ACTION _brand_colors:
IF csp_main_brand.count = '6Count' 
THEN
	brand1_active := TRUE;
ELSE
	brand1_active := FALSE;
END_IF
IF csp_main_brand.count = '8Count' 
THEN
	brand2_active := TRUE;
ELSE
	brand2_active := FALSE;
END_IF
IF csp_main_brand.count = '10Count' 
THEN
	brand3_active := TRUE;
ELSE
	brand3_active := FALSE;
END_IF
IF csp_main_brand.count = '12Count' 
THEN
	brand4_active := TRUE;
ELSE
	brand4_active := FALSE;
END_IF
IF csp_main_brand.count = '16Count2x3' 
THEN
	brand5_active := TRUE;
ELSE
	brand5_active := FALSE;
END_IF
IF csp_main_brand.count = '18Count' 
THEN
	brand6_active := TRUE;
ELSE
	brand6_active := FALSE;
END_IF
IF csp_main_brand.count = '14Count' 
THEN
	brand7_active := TRUE;
ELSE
	brand7_active := FALSE;
END_IF
IF csp_main_brand.count = '16Count2x4' 
THEN
	brand8_active := TRUE;
ELSE
	brand8_active := FALSE;
END_IF
IF csp_main_brand.count = '20Count' 
THEN
	brand9_active := TRUE;
ELSE
	brand9_active := FALSE;
END_IF
IF csp_main_brand.count = '22Count' 
THEN
	brand10_active := TRUE;
ELSE
	brand10_active := FALSE;
END_IF
IF csp_main_brand.count = '24Count' 
THEN
	brand11_active := TRUE;
ELSE
	brand11_active := FALSE;
END_IF
IF csp_main_brand.count = '28Count' 
THEN
	brand12_active := TRUE;
ELSE
	brand12_active := FALSE;
END_IF
IF csp_main_brand.count = '30Count' 
THEN
	brand13_active := TRUE;
ELSE
	brand13_active := FALSE;
END_IF
IF csp_main_brand.count = '32Count' 
THEN
	brand14_active := TRUE;
ELSE
	brand14_active := FALSE;
END_IF
IF csp_main_brand.count = '34Count' 
THEN
	brand15_active := TRUE;
ELSE
	brand15_active := FALSE;
END_IF
IF csp_main_brand.count = '36Count' 
THEN
	brand16_active := TRUE;
ELSE
	brand16_active := FALSE;
END_IF
IF csp_main_brand.count = '44Count' 
THEN
	brand17_active := TRUE;
ELSE
	brand17_active := FALSE;
END_IF
IF csp_main_brand.count = '46Count' 
THEN
	brand18_active := TRUE;
ELSE
	brand18_active := FALSE;
END_IF
IF csp_main_brand.count = '48Count' 
THEN
	brand19_active := TRUE;
ELSE
	brand19_active := FALSE;
END_IF
IF brand1_active 
THEN
	hmi_change_part_eoat_color := RED;
	hmi_change_part_pusher_color := GREEN;
	hmi_change_part_plate_color	:= GREEN;
	hmi_change_part_paddle_color := RED; (* NO COLOR BUT NEEDS VALUE *)
END_IF
IF brand2_active 
THEN
	hmi_change_part_eoat_color := GREEN;
	hmi_change_part_pusher_color := GREEN;
	hmi_change_part_plate_color	:= GREEN;
	hmi_change_part_paddle_color := RED; (* NO COLOR BUT NEEDS VALUE *)
END_IF
IF brand3_active 
THEN
	hmi_change_part_eoat_color := BLUE;
	hmi_change_part_pusher_color := YELLOW;
	hmi_change_part_plate_color	:= YELLOW;
	hmi_change_part_paddle_color := RED; (* NO COLOR BUT NEEDS VALUE *)
END_IF
IF brand4_active 
THEN
	hmi_change_part_eoat_color := BLUE;
	hmi_change_part_pusher_color := YELLOW;
	hmi_change_part_plate_color	:= YELLOW;
	hmi_change_part_paddle_color := RED; (* NO COLOR BUT NEEDS VALUE *)
END_IF
IF brand5_active 
THEN
	hmi_change_part_eoat_color := BLUE;
	hmi_change_part_pusher_color := YELLOW;
	hmi_change_part_plate_color	:= YELLOW;
	hmi_change_part_paddle_color := RED; (* NO COLOR BUT NEEDS VALUE *)
END_IF
IF brand6_active 
THEN
	hmi_change_part_eoat_color := BLUE;
	hmi_change_part_pusher_color := YELLOW;
	hmi_change_part_plate_color	:= YELLOW;
	hmi_change_part_paddle_color := RED; (* NO COLOR BUT NEEDS VALUE *)
END_IF
IF brand7_active 
THEN
	hmi_change_part_eoat_color := YELLOW;
	hmi_change_part_pusher_color := YELLOW;
	hmi_change_part_plate_color	:= YELLOW;
	hmi_change_part_paddle_color := RED; (* NO COLOR BUT NEEDS VALUE *)
END_IF
IF brand8_active 
THEN
	hmi_change_part_eoat_color := YELLOW;
	hmi_change_part_pusher_color := YELLOW;
	hmi_change_part_plate_color	:= YELLOW;
	hmi_change_part_paddle_color := RED; (* NO COLOR BUT NEEDS VALUE *)
END_IF
IF brand9_active 
THEN
	hmi_change_part_eoat_color := YELLOW;
	hmi_change_part_pusher_color := YELLOW;
	hmi_change_part_plate_color	:= YELLOW;
	hmi_change_part_paddle_color := RED; (* NO COLOR BUT NEEDS VALUE *)
END_IF
IF brand10_active 
THEN
	hmi_change_part_eoat_color := YELLOW;
	hmi_change_part_pusher_color := YELLOW;
	hmi_change_part_plate_color	:= YELLOW;
	hmi_change_part_paddle_color := RED; (* NO COLOR BUT NEEDS VALUE *)
END_IF
IF brand11_active 
THEN
	hmi_change_part_eoat_color := YELLOW;
	hmi_change_part_pusher_color := YELLOW;
	hmi_change_part_plate_color	:= YELLOW;
	hmi_change_part_paddle_color := RED; (* NO COLOR BUT NEEDS VALUE *)
END_IF
IF brand12_active 
THEN
	hmi_change_part_eoat_color := WHITE;
	hmi_change_part_pusher_color := WHITE;
	hmi_change_part_plate_color	:= BLACK;
	hmi_change_part_paddle_color := RED; (* NO COLOR BUT NEEDS VALUE *)
END_IF
IF brand13_active 
THEN
	hmi_change_part_eoat_color := WHITE;
	hmi_change_part_pusher_color := WHITE;
	hmi_change_part_plate_color	:= BLACK;
	hmi_change_part_paddle_color := RED; (* NO COLOR BUT NEEDS VALUE *)
END_IF
IF brand14_active 
THEN
	hmi_change_part_eoat_color := WHITE;
	hmi_change_part_pusher_color := WHITE;
	hmi_change_part_plate_color	:= BLACK;
	hmi_change_part_paddle_color := RED; (* NO COLOR BUT NEEDS VALUE *)
END_IF
IF brand15_active 
THEN
	hmi_change_part_eoat_color := BLACK;
	hmi_change_part_pusher_color := BLACK;
	hmi_change_part_plate_color	:= BLACK;
	hmi_change_part_paddle_color := RED; (* NO COLOR BUT NEEDS VALUE *)
END_IF
IF brand16_active 
THEN
	hmi_change_part_eoat_color := BLACK;
	hmi_change_part_pusher_color := BLACK;
	hmi_change_part_plate_color	:= BLACK;
	hmi_change_part_paddle_color := RED; (* NO COLOR BUT NEEDS VALUE *)
END_IF
IF brand17_active 
THEN
	hmi_change_part_eoat_color := ORANGE;
	hmi_change_part_pusher_color := BLACK;
	hmi_change_part_plate_color	:= BLACK;
	hmi_change_part_paddle_color := RED; (* NO COLOR BUT NEEDS VALUE *)
END_IF
IF brand18_active 
THEN
	hmi_change_part_eoat_color := ORANGE;
	hmi_change_part_pusher_color := BLACK;
	hmi_change_part_plate_color	:= BLACK;
	hmi_change_part_paddle_color := RED; (* NO COLOR BUT NEEDS VALUE *)
END_IF
IF brand19_active 
THEN
	hmi_change_part_eoat_color := RED;		//07/08/21 PRS (was ORANGE)
	hmi_change_part_pusher_color := BLACK;
	hmi_change_part_plate_color	:= BLACK;
	hmi_change_part_paddle_color := RED; (* NO COLOR BUT NEEDS VALUE *)
END_IF
END_ACTION

ACTION _handle_messages:
IF	navigate_to_accU_popup
THEN
	process_message_set(
		errorID_1			:= 0,//fbConfigKinGroup.nErrorId,
		errorID_2			:= 0,
		errorID_3			:= 0,
		CONVERSION_this 	:= navigate_custom_screen_aem);
ELSE
	process_message_reset(navigate_custom_screen_aem);
END_IF

IF	trigger_change_parts_incorrect_popup
THEN
	process_message_set(
		errorID_1			:= 0,
		errorID_2			:= 0,
		errorID_3			:= 0,
		CONVERSION_this 	:= change_parts_incorrect_aem);
ELSE
	process_message_reset(change_parts_incorrect_aem);
END_IF
END_ACTION

ACTION _handle_process_test:
;
END_ACTION

ACTION _hmi_management:
CASE hmi_current_accU_step OF
	0:
		hmi_accU_step1_on:= FALSE;
		hmi_accU_step2_on:= FALSE;
		hmi_accU_step3_on:= FALSE;
		hmi_accU_step4_on:= FALSE;
		hmi_accU_step5_on:= FALSE;
		hmi_accU_step6_on:= FALSE;
		hmi_accU_step7_on:= FALSE;
	1:
		hmi_accU_step1_on:= TRUE;
		hmi_accU_step2_on:= FALSE;
		hmi_accU_step3_on:= FALSE;
		hmi_accU_step4_on:= FALSE;
		hmi_accU_step5_on:= FALSE;
		hmi_accU_step6_on:= FALSE;
		hmi_accU_step7_on:= FALSE;
	2:
		hmi_accU_step1_on:= FALSE;
		hmi_accU_step2_on:= TRUE;
		hmi_accU_step3_on:= FALSE;
		hmi_accU_step4_on:= FALSE;
		hmi_accU_step5_on:= FALSE;
		hmi_accU_step6_on:= FALSE;
		hmi_accU_step7_on:= FALSE;
	3:
		hmi_accU_step1_on:= FALSE;
		hmi_accU_step2_on:= FALSE;
		hmi_accU_step3_on:= TRUE;
		hmi_accU_step4_on:= FALSE;
		hmi_accU_step5_on:= FALSE;
		hmi_accU_step6_on:= FALSE;
		hmi_accU_step7_on:= FALSE;
	4:
		hmi_accU_step1_on:= FALSE;
		hmi_accU_step2_on:= FALSE;
		hmi_accU_step3_on:= FALSE;
		hmi_accU_step4_on:= TRUE;
		hmi_accU_step5_on:= FALSE;
		hmi_accU_step6_on:= FALSE;
		hmi_accU_step7_on:= FALSE;
	5:
		hmi_accU_step1_on:= FALSE;
		hmi_accU_step2_on:= FALSE;
		hmi_accU_step3_on:= FALSE;
		hmi_accU_step4_on:= FALSE;
		hmi_accU_step5_on:= TRUE;
		hmi_accU_step6_on:= FALSE;
		hmi_accU_step7_on:= FALSE;
	6:
		hmi_accU_step1_on:= FALSE;
		hmi_accU_step2_on:= FALSE;
		hmi_accU_step3_on:= FALSE;
		hmi_accU_step4_on:= FALSE;
		hmi_accU_step5_on:= FALSE;
		hmi_accU_step6_on:= TRUE;
		hmi_accU_step7_on:= FALSE;
	7:
		hmi_accU_step1_on:= FALSE;
		hmi_accU_step2_on:= FALSE;
		hmi_accU_step3_on:= FALSE;
		hmi_accU_step4_on:= FALSE;
		hmi_accU_step5_on:= FALSE;
		hmi_accU_step6_on:= FALSE;
		hmi_accU_step7_on:= TRUE;
END_CASE

CASE hmi_change_part_eoat_color OF
	RED:
		hmi_change_part_eoat_red_on:= TRUE;
		hmi_change_part_eoat_green_on:= FALSE;
		hmi_change_part_eoat_blue_on:= FALSE;
		hmi_change_part_eoat_yellow_on:= FALSE;
		hmi_change_part_eoat_white_on:= FALSE;
		hmi_change_part_eoat_black_on:= FALSE;
		hmi_change_part_eoat_orange_on:= FALSE;
	GREEN:
		hmi_change_part_eoat_red_on:= FALSE;
		hmi_change_part_eoat_green_on:= TRUE;
		hmi_change_part_eoat_blue_on:= FALSE;
		hmi_change_part_eoat_yellow_on:= FALSE;
		hmi_change_part_eoat_white_on:= FALSE;
		hmi_change_part_eoat_black_on:= FALSE;
		hmi_change_part_eoat_orange_on:= FALSE;
	BLUE:
		hmi_change_part_eoat_red_on:= FALSE;
		hmi_change_part_eoat_green_on:= FALSE;
		hmi_change_part_eoat_blue_on:= TRUE;
		hmi_change_part_eoat_yellow_on:= FALSE;
		hmi_change_part_eoat_white_on:= FALSE;
		hmi_change_part_eoat_black_on:= FALSE;
		hmi_change_part_eoat_orange_on:= FALSE;
	YELLOW:
		hmi_change_part_eoat_red_on:= FALSE;
		hmi_change_part_eoat_green_on:= FALSE;
		hmi_change_part_eoat_blue_on:= FALSE;
		hmi_change_part_eoat_yellow_on:= TRUE;
		hmi_change_part_eoat_white_on:= FALSE;
		hmi_change_part_eoat_black_on:= FALSE;
		hmi_change_part_eoat_orange_on:= FALSE;
	WHITE:
		hmi_change_part_eoat_red_on:= FALSE;
		hmi_change_part_eoat_green_on:= FALSE;
		hmi_change_part_eoat_blue_on:= FALSE;
		hmi_change_part_eoat_yellow_on:= FALSE;
		hmi_change_part_eoat_white_on:= TRUE;
		hmi_change_part_eoat_black_on:= FALSE;
		hmi_change_part_eoat_orange_on:= FALSE;
	BLACK:
		hmi_change_part_eoat_red_on:= FALSE;
		hmi_change_part_eoat_green_on:= FALSE;
		hmi_change_part_eoat_blue_on:= FALSE;
		hmi_change_part_eoat_yellow_on:= FALSE;
		hmi_change_part_eoat_white_on:= FALSE;
		hmi_change_part_eoat_black_on:= TRUE;
		hmi_change_part_eoat_orange_on:= FALSE;
	ORANGE:
		hmi_change_part_eoat_red_on:= FALSE;
		hmi_change_part_eoat_green_on:= FALSE;
		hmi_change_part_eoat_blue_on:= FALSE;
		hmi_change_part_eoat_yellow_on:= FALSE;
		hmi_change_part_eoat_white_on:= FALSE;
		hmi_change_part_eoat_black_on:= FALSE;
		hmi_change_part_eoat_orange_on:= TRUE;
END_CASE

CASE hmi_change_part_pusher_color OF
	GREEN:
		hmi_change_part_pusher_green_on:= TRUE;
		hmi_change_part_pusher_yellow_on:= FALSE;
		hmi_change_part_pusher_white_on:= FALSE;
		hmi_change_part_pusher_black_on:= FALSE;
	YELLOW:
		hmi_change_part_pusher_green_on:= FALSE;
		hmi_change_part_pusher_yellow_on:= TRUE;
		hmi_change_part_pusher_white_on:= FALSE;
		hmi_change_part_pusher_black_on:= FALSE;
	WHITE:
		hmi_change_part_pusher_green_on:= FALSE;
		hmi_change_part_pusher_yellow_on:= FALSE;
		hmi_change_part_pusher_white_on:= TRUE;
		hmi_change_part_pusher_black_on:= FALSE;
	BLACK:
		hmi_change_part_pusher_green_on:= FALSE;
		hmi_change_part_pusher_yellow_on:= FALSE;
		hmi_change_part_pusher_white_on:= FALSE;
		hmi_change_part_pusher_black_on:= TRUE;
END_CASE

CASE hmi_change_part_plate_color OF
	GREEN:
		hmi_change_part_plate_green_on:= TRUE;
		hmi_change_part_plate_yellow_on:= FALSE;
		hmi_change_part_plate_black_on:= FALSE;
	YELLOW:
		hmi_change_part_plate_green_on:= FALSE;
		hmi_change_part_plate_yellow_on:= TRUE;
		hmi_change_part_plate_black_on:= FALSE;
	BLACK:
		hmi_change_part_plate_green_on:= FALSE;
		hmi_change_part_plate_yellow_on:= FALSE;
		hmi_change_part_plate_black_on:= TRUE;
END_CASE

CASE hmi_change_part_paddle_color OF
	NO_COLOR:
		//FUTURE PLACEHOLDER
END_CASE

	hmi_graphic_object_set_status(
		status  			:= SEL(machine_size_complete, HMI_OBJECT_STATUS_INVISIBLE, HMI_OBJECT_STATUS_ON),
		CONVERSION_this    	:= hmi_brand_status_color_hgos);
	
	hmi_graphic_object_set_status(
		status  			:= SEL(machine_size_complete, HMI_OBJECT_STATUS_ON, HMI_OBJECT_STATUS_INVISIBLE),
		CONVERSION_this    	:= hmi_brand_status_bad_color_hgos);
	
	hmi_graphic_object_set_status(
        status  			:= SEL(hmi_accU_step1_on, HMI_OBJECT_STATUS_INVISIBLE, HMI_OBJECT_STATUS_ON),
        CONVERSION_this     := hmi_accU_step1_on_hgos);
		
	hmi_graphic_object_set_status(
        status  			:= SEL(hmi_accU_step1_on, HMI_OBJECT_STATUS_ON, HMI_OBJECT_STATUS_INVISIBLE),
        CONVERSION_this     := hmi_accU_step1_off_hgos);
		
	hmi_graphic_object_set_status(
        status  			:= SEL(hmi_accU_step2_on, HMI_OBJECT_STATUS_INVISIBLE, HMI_OBJECT_STATUS_ON),
        CONVERSION_this     := hmi_accU_step2_on_hgos);
		
	hmi_graphic_object_set_status(
        status  			:= SEL(hmi_accU_step2_on, HMI_OBJECT_STATUS_ON, HMI_OBJECT_STATUS_INVISIBLE),
        CONVERSION_this     := hmi_accU_step2_off_hgos);
		
	hmi_graphic_object_set_status(
        status  			:= SEL(hmi_accU_step3_on, HMI_OBJECT_STATUS_INVISIBLE, HMI_OBJECT_STATUS_ON),
        CONVERSION_this     := hmi_accU_step3_on_hgos);
		
	hmi_graphic_object_set_status(
        status  			:= SEL(hmi_accU_step3_on, HMI_OBJECT_STATUS_ON, HMI_OBJECT_STATUS_INVISIBLE),
        CONVERSION_this     := hmi_accU_step3_off_hgos);
		
	hmi_graphic_object_set_status(
        status  			:= SEL(hmi_accU_step4_on, HMI_OBJECT_STATUS_INVISIBLE, HMI_OBJECT_STATUS_ON),
        CONVERSION_this     := hmi_accU_step4_on_hgos);
		
	hmi_graphic_object_set_status(
		status  			:= SEL(hmi_accU_step4_on, HMI_OBJECT_STATUS_ON, HMI_OBJECT_STATUS_INVISIBLE),
        CONVERSION_this     := hmi_accU_step4_off_hgos);
		
	hmi_graphic_object_set_status(
        status  			:= SEL(hmi_accU_step5_on, HMI_OBJECT_STATUS_INVISIBLE, HMI_OBJECT_STATUS_ON),
        CONVERSION_this     := hmi_accU_step5_on_hgos);
		
	hmi_graphic_object_set_status(
        status  			:= SEL(hmi_accU_step5_on, HMI_OBJECT_STATUS_ON, HMI_OBJECT_STATUS_INVISIBLE),
        CONVERSION_this     := hmi_accU_step5_off_hgos);
		
	hmi_graphic_object_set_status(
        status  			:= SEL(hmi_accU_step6_on, HMI_OBJECT_STATUS_INVISIBLE, HMI_OBJECT_STATUS_ON),
        CONVERSION_this     := hmi_accU_step6_on_hgos);
		
	hmi_graphic_object_set_status(
        status  			:= SEL(hmi_accU_step6_on, HMI_OBJECT_STATUS_ON, HMI_OBJECT_STATUS_INVISIBLE),
        CONVERSION_this     := hmi_accU_step6_off_hgos);
		
	hmi_graphic_object_set_status(
        status  			:= SEL(hmi_accU_step7_on, HMI_OBJECT_STATUS_INVISIBLE, HMI_OBJECT_STATUS_ON),
        CONVERSION_this     := hmi_accU_step7_on_hgos);
	
	hmi_graphic_object_set_status(
        status  			:= SEL(hmi_accU_step7_on, HMI_OBJECT_STATUS_ON, HMI_OBJECT_STATUS_INVISIBLE),
        CONVERSION_this     := hmi_accU_step7_off_hgos);

	//Change Part EOAT
	hmi_graphic_object_set_status(
        status  			:= SEL(hmi_change_part_eoat_red_on, HMI_OBJECT_STATUS_INVISIBLE, HMI_OBJECT_STATUS_ON),
        CONVERSION_this     := hmi_change_part_eoat_red_hgos);
		
	hmi_graphic_object_set_status(
        status  			:= SEL(hmi_change_part_eoat_green_on, HMI_OBJECT_STATUS_INVISIBLE, HMI_OBJECT_STATUS_ON),
        CONVERSION_this     := hmi_change_part_eoat_green_hgos);
		
	hmi_graphic_object_set_status(
        status  			:= SEL(hmi_change_part_eoat_blue_on, HMI_OBJECT_STATUS_INVISIBLE, HMI_OBJECT_STATUS_ON),
        CONVERSION_this     := hmi_change_part_eoat_blue_hgos);
		
	hmi_graphic_object_set_status(
        status  			:= SEL(hmi_change_part_eoat_yellow_on, HMI_OBJECT_STATUS_INVISIBLE, HMI_OBJECT_STATUS_ON),
        CONVERSION_this     := hmi_change_part_eoat_yellow_hgos);
	
	hmi_graphic_object_set_status(
        status  			:= SEL(hmi_change_part_eoat_white_on, HMI_OBJECT_STATUS_INVISIBLE, HMI_OBJECT_STATUS_ON),
        CONVERSION_this     := hmi_change_part_eoat_white_hgos);
		
	hmi_graphic_object_set_status(
        status  			:= SEL(hmi_change_part_eoat_black_on, HMI_OBJECT_STATUS_INVISIBLE, HMI_OBJECT_STATUS_ON),
        CONVERSION_this     := hmi_change_part_eoat_black_hgos);
		
	hmi_graphic_object_set_status(
        status  			:= SEL(hmi_change_part_eoat_orange_on, HMI_OBJECT_STATUS_INVISIBLE, HMI_OBJECT_STATUS_ON),
        CONVERSION_this     := hmi_change_part_eoat_orange_hgos);
		
	hmi_graphic_object_set_status(
        status  			:= SEL(hmi_change_part_eoat_checkbox_on, HMI_OBJECT_STATUS_INVISIBLE, HMI_OBJECT_STATUS_ON),
        CONVERSION_this     := hmi_change_part_eoat_checkbox_hgos);
		
	//Change Part Pusher
	hmi_graphic_object_set_status(
        status  			:= SEL(hmi_change_part_pusher_green_on, HMI_OBJECT_STATUS_INVISIBLE, HMI_OBJECT_STATUS_ON),
        CONVERSION_this     := hmi_change_part_pusher_green_hgos);
		
	hmi_graphic_object_set_status(
        status  			:= SEL(hmi_change_part_pusher_yellow_on, HMI_OBJECT_STATUS_INVISIBLE, HMI_OBJECT_STATUS_ON),
        CONVERSION_this     := hmi_change_part_pusher_yellow_hgos);
		
	hmi_graphic_object_set_status(
        status  			:= SEL(hmi_change_part_pusher_white_on, HMI_OBJECT_STATUS_INVISIBLE, HMI_OBJECT_STATUS_ON),
        CONVERSION_this     := hmi_change_part_pusher_white_hgos);
		
	hmi_graphic_object_set_status(
        status  			:= SEL(hmi_change_part_pusher_black_on, HMI_OBJECT_STATUS_INVISIBLE, HMI_OBJECT_STATUS_ON),
        CONVERSION_this     := hmi_change_part_pusher_black_hgos);
		
	hmi_graphic_object_set_status(
        status  			:= SEL(hmi_change_part_pusher_checkbox_on, HMI_OBJECT_STATUS_INVISIBLE, HMI_OBJECT_STATUS_ON),
        CONVERSION_this     := hmi_change_part_pusher_checkbox_hgos);
		
	//Change Part Plate
	hmi_graphic_object_set_status(
        status  			:= SEL(hmi_change_part_plate_green_on, HMI_OBJECT_STATUS_INVISIBLE, HMI_OBJECT_STATUS_ON),
        CONVERSION_this     := hmi_change_part_plate_green_hgos);
		
	hmi_graphic_object_set_status(
        status  			:= SEL(hmi_change_part_plate_yellow_on, HMI_OBJECT_STATUS_INVISIBLE, HMI_OBJECT_STATUS_ON),
        CONVERSION_this     := hmi_change_part_plate_yellow_hgos);
		
	hmi_graphic_object_set_status(
        status  			:= SEL(hmi_change_part_plate_black_on, HMI_OBJECT_STATUS_INVISIBLE, HMI_OBJECT_STATUS_ON),
        CONVERSION_this     := hmi_change_part_plate_black_hgos);
		
	hmi_graphic_object_set_status(
        status  			:= SEL(hmi_change_part_plate_checkbox_on, HMI_OBJECT_STATUS_INVISIBLE, HMI_OBJECT_STATUS_ON),
        CONVERSION_this     := hmi_change_part_plate_checkbox_hgos);
	
	//Change Part Paddles
	hmi_graphic_object_set_status(
        status  			:= SEL(hmi_change_part_paddle_checkbox_on, HMI_OBJECT_STATUS_INVISIBLE, HMI_OBJECT_STATUS_ON),
        CONVERSION_this     := hmi_change_part_paddle_checkbox_hgos);
END_ACTION

ACTION _in_position:
IF (csp_case_main_statistics.is_empty
	AND csp_transfer_main_statistics.is_empty 
	AND NOT digital_input_is_active(csp_case_feed_magazine_ls_pusher.retracted_di)
	AND NOT digital_input_is_active(csp_case_feed_magazine_ls_pusherTilt.upstream_di)
	AND NOT digital_input_is_active(csp_case_feed_magazine_os_pusher.retracted_di)
	AND NOT digital_input_is_active(csp_case_feed_magazine_os_pusherTilt.upstream_di)
	AND NOT digital_input_is_active(csp_case_feed_magazine_level_zonemin.di)
	AND NOT digital_input_is_active(csp_case_feed_magazine_level_zonelow.di)
	AND NOT digital_input_is_active(csp_case_feed_magazine_level_zone1.di)
	AND NOT digital_input_is_active(csp_case_feed_magazine_level_zone2.di)
	AND NOT digital_input_is_active(csp_case_feed_magazine_level_zone3.di))
	OR manual_empty
THEN
	machine_empty := TRUE;
ELSE
	machine_empty := FALSE;
END_IF

IF (csp_case_tr_squaring_ls_leading.in_accu_safe_pos)
    AND (csp_case_tr_squaring_ls_trailing.in_accu_safe_pos)
    AND (csp_case_tr_squaring_os_leading.in_accu_safe_pos)
    AND (csp_case_tr_squaring_os_trailing.in_accu_safe_pos)
    AND (csp_case_closing_os_horizontal.in_accu_safe_pos)
    AND (csp_case_closing_os_upper.in_accu_safe_pos)
    AND (csp_case_closing_os_lower.in_accu_safe_pos)
    AND (csp_case_closing_ls_horizontal.in_accu_safe_pos)
    AND (csp_case_closing_ls_upper.in_accu_safe_pos)
    AND (csp_case_closing_ls_lower.in_accu_safe_pos)
    AND (csp_case_fc_ls_lower_follower.in_accu_safe_pos)
    AND (csp_case_fc_ls_lower_spreader.in_accu_safe_pos)
    AND (csp_case_fc_ls_upper_follower.in_accu_safe_pos)
    AND (csp_case_fc_ls_upper_leadingMinorCloser.in_accu_safe_pos)
    AND (csp_case_fc_ls_upper_spreader.in_accu_safe_pos)
    AND (csp_case_fc_os_lower_follower.in_accu_safe_pos)
    AND (csp_case_fc_os_lower_spreader.in_accu_safe_pos)
    AND (csp_case_fc_os_upper_follower.in_accu_safe_pos)
    AND (csp_case_fc_os_upper_spreader.in_accu_safe_pos)
    AND (csp_case_feed_shuttle_vertical.in_accu_safe_pos)
    AND (csp_case_loader_guide_downstream.in_accu_safe_pos)
    AND (csp_case_loader_guide_length.in_accu_safe_pos)
    AND (csp_case_loader_guide_upstream.in_accu_safe_pos)
    AND (csp_case_loader_pusher.in_accu_safe_pos)
	AND (csp_case_feed_kinematic_x.in_accu_safe_pos)
	AND (csp_case_feed_kinematic_y.in_accu_safe_pos)
	AND (csp_case_feed_kinematic_tilt.in_accu_safe_pos) 
THEN
    Case_Motors_Safe_accU := TRUE;
ELSE
    Case_Motors_Safe_accU := FALSE;   
END_IF

	
IF csp_case_feed_shuttle_accU_depth.in_position
	AND csp_case_transport_accU_depth.in_position
	AND csp_case_feed_reject_accU_depth.in_position
THEN
	test_in_position := TRUE;
ELSE
	test_in_position := FALSE;
END_IF

//INSERT IF STATEMENT HERE FOR WHICH MOTORS BELONG TO WHICH GROUP

//Group 1 Motors in Position
IF 	csp_case_transport_accU_depth.in_position
	AND csp_case_feed_shuttle_accU_depth.in_position
	AND csp_case_feed_magazine_accU_lsDepth.in_position
	AND csp_case_feed_magazine_accU_osDepth.in_position
	AND csp_case_feed_reject_accU_depth.in_position
	AND csp_transfer_infeed_accU_depth.in_position
	AND csp_transfer_infeed_accU_waterfallAdjust.in_position
	AND csp_transfer_accumulator_accU_depth.in_position
	AND csp_transfer_accumulator_accU_convDepth.in_position
	AND csp_case_tr_accU_depth.in_position
THEN
	Group_1_motors_in_position := TRUE;
ELSE
	Group_1_motors_in_position := FALSE;
END_IF

//Group 2 Motors in Position
IF 	csp_case_loader_guide_accU_width.in_position
	AND csp_case_glue_os_accU_width.in_position
	AND csp_case_glue_os_accU_upperPosition.in_position
	AND csp_case_glue_os_accU_lowerPosition.in_position
	AND csp_case_glue_ls_accU_upperPosition.in_position
	AND csp_case_glue_ls_accU_lowerPosition.in_position
	AND csp_case_tr_accU_os_width.in_position
	AND csp_case_tr_accU_ls_width.in_position
THEN
	Group_2_motors_in_position := TRUE;
ELSE
	Group_2_motors_in_position := FALSE;
END_IF

IF Case_Motors_In_New_Accu_Pos //AND Transfer_Motors_In_New_Accu_Pos
THEN
	Motion_motors_in_position := TRUE;
ELSE
	Motion_motors_in_position := FALSE;
END_IF


IF 	ABS(csp_case_closing_os_horizontal.axis.actual_position - csp_case_closing_os_horizontal.accu_safe_pos) < csp_case_closing_os_horizontal.accu_tolerance
	AND ABS(csp_case_closing_ls_horizontal.axis.actual_position - csp_case_closing_ls_horizontal.accu_safe_pos) < csp_case_closing_ls_horizontal.accu_tolerance
THEN
	closing_horizontal_safe := TRUE;
ELSE
	closing_horizontal_safe := FALSE;
END_IF


(* Acc U Change indicators on Acc U Change Motor page *)
	
	hmi_graphic_object_set_status(
        status  			:= SEL(csp_case_transport_accU_depth.in_position, HMI_OBJECT_STATUS_INVISIBLE, HMI_OBJECT_STATUS_ON),
        CONVERSION_this     := hmi_in_position_transport_depth_on_hgos);
		
	hmi_graphic_object_set_status(
        status  			:= SEL(csp_case_transport_accU_depth.in_position, HMI_OBJECT_STATUS_ON, HMI_OBJECT_STATUS_INVISIBLE),
        CONVERSION_this     := hmi_in_position_transport_depth_off_hgos);
	
	hmi_graphic_object_set_status(
        status  			:= SEL(csp_case_feed_shuttle_accU_depth.in_position, HMI_OBJECT_STATUS_INVISIBLE, HMI_OBJECT_STATUS_ON),
        CONVERSION_this     := hmi_in_position_shuttle_depth_on_hgos);
		
	hmi_graphic_object_set_status(
        status  			:= SEL(csp_case_feed_shuttle_accU_depth.in_position, HMI_OBJECT_STATUS_ON, HMI_OBJECT_STATUS_INVISIBLE),
        CONVERSION_this     := hmi_in_position_shuttle_depth_off_hgos);

 	hmi_graphic_object_set_status(
        status  			:= SEL(csp_case_feed_magazine_accU_lsDepth.in_position, HMI_OBJECT_STATUS_INVISIBLE, HMI_OBJECT_STATUS_ON),
        CONVERSION_this     := hmi_in_position_magazine_ls_depth_on_hgos);
		
	hmi_graphic_object_set_status(
        status  			:= SEL(csp_case_feed_magazine_accU_lsDepth.in_position, HMI_OBJECT_STATUS_ON, HMI_OBJECT_STATUS_INVISIBLE),
        CONVERSION_this     := hmi_in_position_magazine_ls_depth_off_hgos);
		
	hmi_graphic_object_set_status(
        status  			:= SEL(csp_case_feed_magazine_accU_osDepth.in_position, HMI_OBJECT_STATUS_INVISIBLE, HMI_OBJECT_STATUS_ON),
        CONVERSION_this     := hmi_in_position_magazine_os_depth_on_hgos);
		
	hmi_graphic_object_set_status(
        status  			:= SEL(csp_case_feed_magazine_accU_osDepth.in_position, HMI_OBJECT_STATUS_ON, HMI_OBJECT_STATUS_INVISIBLE),
        CONVERSION_this     := hmi_in_position_magazine_os_depth_off_hgos);
	
	hmi_graphic_object_set_status(
        status  			:= SEL(csp_case_feed_reject_accU_depth.in_position, HMI_OBJECT_STATUS_INVISIBLE, HMI_OBJECT_STATUS_ON),
        CONVERSION_this     := hmi_in_position_discharge_os_depth_on_hgos);
		
	hmi_graphic_object_set_status(
        status  			:= SEL(csp_case_feed_reject_accU_depth.in_position, HMI_OBJECT_STATUS_ON, HMI_OBJECT_STATUS_INVISIBLE),
        CONVERSION_this     := hmi_in_position_discharge_os_depth_off_hgos);
	
	hmi_graphic_object_set_status(
        status  			:= SEL(csp_transfer_infeed_accU_depth.in_position, HMI_OBJECT_STATUS_INVISIBLE, HMI_OBJECT_STATUS_ON),
        CONVERSION_this     := hmi_in_position_transfer_infeed_depth_on_hgos);
		
	hmi_graphic_object_set_status(
        status  			:= SEL(csp_transfer_infeed_accU_depth.in_position, HMI_OBJECT_STATUS_ON, HMI_OBJECT_STATUS_INVISIBLE),
        CONVERSION_this     := hmi_in_position_transfer_infeed_depth_off_hgos);	
		
	hmi_graphic_object_set_status(
        status  			:= SEL(csp_transfer_infeed_accU_waterfallAdjust.in_position, HMI_OBJECT_STATUS_INVISIBLE, HMI_OBJECT_STATUS_ON),
        CONVERSION_this     := hmi_in_position_waterfall_on_hgos);
		
	hmi_graphic_object_set_status(
        status  			:= SEL(csp_transfer_infeed_accU_waterfallAdjust.in_position, HMI_OBJECT_STATUS_ON, HMI_OBJECT_STATUS_INVISIBLE),
        CONVERSION_this     := hmi_in_position_waterfall_off_hgos);	
	 
	hmi_graphic_object_set_status(
        status  			:= SEL(csp_transfer_accumulator_accU_depth.in_position, HMI_OBJECT_STATUS_INVISIBLE, HMI_OBJECT_STATUS_ON),
        CONVERSION_this     := hmi_in_position_accumulator_depth_on_hgos);
		
	hmi_graphic_object_set_status(
        status  			:= SEL(csp_transfer_accumulator_accU_depth.in_position, HMI_OBJECT_STATUS_ON, HMI_OBJECT_STATUS_INVISIBLE),
        CONVERSION_this     := hmi_in_position_accumulator_depth_off_hgos);	
		
	hmi_graphic_object_set_status(
        status  			:= SEL(csp_transfer_accumulator_accU_convDepth.in_position, HMI_OBJECT_STATUS_INVISIBLE, HMI_OBJECT_STATUS_ON),
        CONVERSION_this     := hmi_in_position_accumulator_conv_depth_on_hgos);
		
	hmi_graphic_object_set_status(
        status  			:= SEL(csp_transfer_accumulator_accU_convDepth.in_position, HMI_OBJECT_STATUS_ON, HMI_OBJECT_STATUS_INVISIBLE),
        CONVERSION_this     := hmi_in_position_accumulator_conv_depth_off_hgos);		

	hmi_graphic_object_set_status(
        status  			:= SEL(csp_case_tr_accU_depth.in_position, HMI_OBJECT_STATUS_INVISIBLE, HMI_OBJECT_STATUS_ON),
        CONVERSION_this     := hmi_in_position_top_rail_depth_on_hgos);
		
	hmi_graphic_object_set_status(
        status  			:= SEL(csp_case_tr_accU_depth.in_position, HMI_OBJECT_STATUS_ON, HMI_OBJECT_STATUS_INVISIBLE),
        CONVERSION_this     := hmi_in_position_top_rail_depth_off_hgos);		

	

//Group 2 Motors in Position Acc U Change motor indicators
	hmi_graphic_object_set_status(
        status  			:= SEL(csp_case_loader_guide_accU_width.in_position, HMI_OBJECT_STATUS_INVISIBLE, HMI_OBJECT_STATUS_ON),
        CONVERSION_this     := hmi_in_position_loader_guide_width_on_hgos);
		
	hmi_graphic_object_set_status(
        status  			:= SEL(csp_case_loader_guide_accU_width.in_position, HMI_OBJECT_STATUS_ON, HMI_OBJECT_STATUS_INVISIBLE),
        CONVERSION_this     := hmi_in_position_loader_guide_width_off_hgos);	
	
	hmi_graphic_object_set_status(
        status  			:= SEL(csp_case_glue_os_accU_width.in_position, HMI_OBJECT_STATUS_INVISIBLE, HMI_OBJECT_STATUS_ON),
        CONVERSION_this     := hmi_in_position_glue_os_width_on_hgos);
		
	hmi_graphic_object_set_status(
        status  			:= SEL(csp_case_glue_os_accU_width.in_position, HMI_OBJECT_STATUS_ON, HMI_OBJECT_STATUS_INVISIBLE),
        CONVERSION_this     := hmi_in_position_glue_os_width_off_hgos);	
		
	hmi_graphic_object_set_status(
        status  			:= SEL(csp_case_glue_os_accU_upperPosition.in_position, HMI_OBJECT_STATUS_INVISIBLE, HMI_OBJECT_STATUS_ON),
        CONVERSION_this     := hmi_in_position_glue_os_upper_on_hgos);
		
	hmi_graphic_object_set_status(
        status  			:= SEL(csp_case_glue_os_accU_upperPosition.in_position, HMI_OBJECT_STATUS_ON, HMI_OBJECT_STATUS_INVISIBLE),
        CONVERSION_this     := hmi_in_position_glue_os_upper_off_hgos);	
		
	hmi_graphic_object_set_status(
        status  			:= SEL(csp_case_glue_os_accU_lowerPosition.in_position, HMI_OBJECT_STATUS_INVISIBLE, HMI_OBJECT_STATUS_ON),
        CONVERSION_this     := hmi_in_position_glue_os_lower_on_hgos);
		
	hmi_graphic_object_set_status(
        status  			:= SEL(csp_case_glue_os_accU_lowerPosition.in_position, HMI_OBJECT_STATUS_ON, HMI_OBJECT_STATUS_INVISIBLE),
        CONVERSION_this     := hmi_in_position_glue_os_lower_off_hgos);	
	
	hmi_graphic_object_set_status(
        status  			:= SEL(csp_case_glue_ls_accU_upperPosition.in_position, HMI_OBJECT_STATUS_INVISIBLE, HMI_OBJECT_STATUS_ON),
        CONVERSION_this     := hmi_in_position_glue_ls_upper_on_hgos);
		
	hmi_graphic_object_set_status(
        status  			:= SEL(csp_case_glue_ls_accU_upperPosition.in_position, HMI_OBJECT_STATUS_ON, HMI_OBJECT_STATUS_INVISIBLE),
        CONVERSION_this     := hmi_in_position_glue_ls_upper_off_hgos);	
		
	hmi_graphic_object_set_status(
        status  			:= SEL(csp_case_glue_ls_accU_lowerPosition.in_position, HMI_OBJECT_STATUS_INVISIBLE, HMI_OBJECT_STATUS_ON),
        CONVERSION_this     := hmi_in_position_glue_ls_lower_on_hgos);
		
	hmi_graphic_object_set_status(
        status  			:= SEL(csp_case_glue_ls_accU_lowerPosition.in_position, HMI_OBJECT_STATUS_ON, HMI_OBJECT_STATUS_INVISIBLE),
        CONVERSION_this     := hmi_in_position_glue_ls_lower_off_hgos);	
	
	hmi_graphic_object_set_status(
        status  			:= SEL(csp_case_tr_accU_os_width.in_position, HMI_OBJECT_STATUS_INVISIBLE, HMI_OBJECT_STATUS_ON),
        CONVERSION_this     := hmi_in_position_top_rail_os_width_on_hgos);
		
	hmi_graphic_object_set_status(
        status  			:= SEL(csp_case_tr_accU_os_width.in_position, HMI_OBJECT_STATUS_ON, HMI_OBJECT_STATUS_INVISIBLE),
        CONVERSION_this     := hmi_in_position_top_rail_os_width_off_hgos);	


	hmi_graphic_object_set_status(
        status  			:= SEL(csp_case_tr_accU_ls_width.in_position, HMI_OBJECT_STATUS_INVISIBLE, HMI_OBJECT_STATUS_ON),
        CONVERSION_this     := hmi_in_position_top_rail_ls_width_on_hgos);
		
	hmi_graphic_object_set_status(
        status  			:= SEL(csp_case_tr_accU_ls_width.in_position, HMI_OBJECT_STATUS_ON, HMI_OBJECT_STATUS_INVISIBLE),
        CONVERSION_this     := hmi_in_position_top_rail_ls_width_off_hgos);
END_ACTION

ACTION _mode_manager:
IF process_mode_req_is_pending(prc)
THEN
    process_apply_mode_req_first_step(prc);
    CASE process_get_mode(prc) OF
        MODE_TO_ABSENT:
			;
        MODE_TO_INACTIVE:
			;
        MODE_TO_TEST:
			;
        MODE_TO_OPERATIONAL:
			;
    END_CASE
    process_apply_mode_req_second_step(prc);
END_IF
END_ACTION

ACTION _object_manager:
IF objects_initialization()
THEN
	sub_process_init(
		object_name					:= 'csp_main_accuChange.prc', 
		process						:= csp_main.prc, 
		CONVERSION_this				:= prc);
		
	prc_path 						:= process_get_path(prc);
	
	process_message_init(
		object_name					:= CONCAT(prc_path, '_navigate_custom_screen_aem'), 
		behaviour					:= MESSAGE_BEHAVIOUR_STATE,
		reset_timeout				:= 0,
		disableable					:= FALSE,
		individual_reset			:= FALSE,
		machine_reaction			:= MACHINE_REACTION_NO_STOP,
		typology					:= MESSAGE_TYPOLOGY_OBLIGATION,
		process						:= prc,
		CONVERSION_this				:= navigate_custom_screen_aem);
		
	process_message_init(
		object_name					:= CONCAT(prc_path, '_change_parts_incorrect_aem'), 
		behaviour					:= MESSAGE_BEHAVIOUR_STATE,
		reset_timeout				:= 0,
		disableable					:= FALSE,
		individual_reset			:= FALSE,
		machine_reaction			:= MACHINE_REACTION_NO_STOP,
		typology					:= MESSAGE_TYPOLOGY_OBLIGATION,
		process						:= prc,
		CONVERSION_this				:= change_parts_incorrect_aem);		
		
	timer_init(
		object_name					:= CONCAT(prc_path, '_RFID_read_write_tmr'),
		process						:= prc,
		CONVERSION_this				:= RFID_read_write_tmr);
	
	motorization_conditioner_init(
		object_name					:=	CONCAT(prc_path, 'all_in_position_motcond'),
		velocity_limit				:=	0.0,
		velocity_limit_active		:=	FALSE,
		idle_handshake_active		:=	FALSE,
		execute_handshake_active	:=	TRUE,
		hold_handshake_active		:=	FALSE,
		suspend_handshake_active	:=	FALSE,
		complete_handshake_active	:=	FALSE,
		abort_handshake_active		:=	FALSE,
		stop_handshake_active		:=	FALSE,
		origin						:=	MOTORIZATION_CONDITIONER_ORIGIN_INTERNAL,
		manager						:=	csp_main_motorization_manager.motm,
		process						:=	prc,
		CONVERSION_this				:=	all_in_position_motcond);
		
		
	motorization_conditioner_init(
		object_name					:=	CONCAT(prc_path, '_eoat_rfid_checked_motcond'),
		velocity_limit				:=	0.0,
		velocity_limit_active		:=	FALSE,
		idle_handshake_active		:=	FALSE,
		execute_handshake_active	:=	TRUE,
		hold_handshake_active		:=	FALSE,
		suspend_handshake_active	:=	FALSE,
		complete_handshake_active	:=	FALSE,
		abort_handshake_active		:=	FALSE,
		stop_handshake_active		:=	FALSE,
		origin						:=	MOTORIZATION_CONDITIONER_ORIGIN_INTERNAL,
		manager						:=	csp_main_motorization_manager.motm,
		process						:=	prc,
		CONVERSION_this				:=	eoat_rfid_checked_motcond);
		
	motorization_conditioner_init(
		object_name					:=	CONCAT(prc_path, '_loader_pusher_rfid_checked_motcond'),
		velocity_limit				:=	0.0,
		velocity_limit_active		:=	FALSE,
		idle_handshake_active		:=	FALSE,
		execute_handshake_active	:=	TRUE,
		hold_handshake_active		:=	FALSE,
		suspend_handshake_active	:=	FALSE,
		complete_handshake_active	:=	FALSE,
		abort_handshake_active		:=	FALSE,
		stop_handshake_active		:=	FALSE,
		origin						:=	MOTORIZATION_CONDITIONER_ORIGIN_INTERNAL,
		manager						:=	csp_main_motorization_manager.motm,
		process						:=	prc,
		CONVERSION_this				:=	loader_pusher_rfid_checked_motcond);
		
	motorization_conditioner_init(
		object_name					:=	CONCAT(prc_path, '_loader_plate_rfid_checked_motcond'),
		velocity_limit				:=	0.0,
		velocity_limit_active		:=	FALSE,
		idle_handshake_active		:=	FALSE,
		execute_handshake_active	:=	TRUE,
		hold_handshake_active		:=	FALSE,
		suspend_handshake_active	:=	FALSE,
		complete_handshake_active	:=	FALSE,
		abort_handshake_active		:=	FALSE,
		stop_handshake_active		:=	FALSE,
		origin						:=	MOTORIZATION_CONDITIONER_ORIGIN_INTERNAL,
		manager						:=	csp_main_motorization_manager.motm,
		process						:=	prc,
		CONVERSION_this				:=	loader_plate_rfid_checked_motcond);
		
		
	boolean_init(
		object_name:= CONCAT(prc_path, '_motors_in_safe_pos_boolean'), 
		process:= prc, 
		CONVERSION_this:= motors_in_safe_pos_boolean);
		
	digital_check_and_message_init(
		object_name:= CONCAT(prc_path, '_stop_machine_for_change_parts_dchk'), 
		alarm_if_input_off:= FALSE, 
		alarm_delay:= 0, 
		enabled_at_powerup:= TRUE, 
		individual_reset:= FALSE, 
		machine_reaction:= MACHINE_REACTION_NORMAL_STOP, 
		typology:= MESSAGE_TYPOLOGY_ABNORMAL, 
		process:= prc, 
		CONVERSION_this:= stop_machine_for_change_parts_dchk);
	
	digital_check_add_boolean(
		boolean:= motors_in_safe_pos_boolean, 
		CONVERSION_this:= stop_machine_for_change_parts_dchk);
	
	
		
	process_message_init(
        object_name:= CONCAT(prc_path, '_change_part_eoat_wrong'),
        behaviour:= MESSAGE_BEHAVIOUR_STATE,
        reset_timeout:= 0,
        disableable:= TRUE,
        individual_reset:= FALSE,
        machine_reaction:= MACHINE_REACTION_NORMAL_STOP, 
        typology:=  MESSAGE_TYPOLOGY_ABNORMAL,
        process:= prc,
        CONVERSION_this:= change_part_eoat_wrong);
		
	process_message_init(
        object_name:= CONCAT(prc_path, '_change_part_pusher_wrong'),
        behaviour:= MESSAGE_BEHAVIOUR_STATE,
        reset_timeout:= 0,
        disableable:= TRUE,
        individual_reset:= FALSE,
        machine_reaction:= MACHINE_REACTION_NORMAL_STOP,
        typology:=  MESSAGE_TYPOLOGY_ABNORMAL, 
        process:= prc,
        CONVERSION_this:= change_part_pusher_wrong);
		
	process_message_init(
        object_name:= CONCAT(prc_path, '_change_part_plate_wrong'),
        behaviour:= MESSAGE_BEHAVIOUR_STATE,
        reset_timeout:= 0,
        disableable:= TRUE,
        individual_reset:= FALSE,
        machine_reaction:= MACHINE_REACTION_NORMAL_STOP,
        typology:=  MESSAGE_TYPOLOGY_ABNORMAL, 
        process:= prc,
        CONVERSION_this:= change_part_plate_wrong);
		
	process_message_init(
        object_name:= CONCAT(prc_path, '_change_part_paddles_wrong'),
        behaviour:= MESSAGE_BEHAVIOUR_STATE,
        reset_timeout:= 0,
        disableable:= TRUE,
        individual_reset:= FALSE,
        machine_reaction:= MACHINE_REACTION_NORMAL_STOP, 
        typology:=  MESSAGE_TYPOLOGY_ABNORMAL, 
        process:= prc,
        CONVERSION_this:= change_part_paddles_wrong);
		
	//HMI custom page variable management	
	command_button_init(
	    object_name 				:= CONCAT(prc_path, '_hmi_toggle_cbtn'),
	    process 					:= prc,
	    CONVERSION_this 			:= hmi_toggle_cbtn);
		
	command_button_init(
	    object_name 				:= CONCAT(prc_path, '_manual_empty_cbtn'),
	    process 					:= prc,
	    CONVERSION_this 			:= manual_empty_cbtn);
		
	command_button_init(
	    object_name 				:= CONCAT(prc_path, '_RFID_Setup_read_cbtn'),
	    process 					:= prc,
	    CONVERSION_this 			:= RFID_Setup_read_cbtn);
		
	command_button_init(
	    object_name 				:= CONCAT(prc_path, '_RFID_Setup_write_cbtn'),
	    process 					:= prc,
	    CONVERSION_this 			:= RFID_Setup_write_cbtn);
	
	command_button_init(
	    object_name 				:= CONCAT(prc_path, '_brand_change_request_cbtn'),
	    process 					:= prc,
	    CONVERSION_this 			:= brand_change_request_cbtn);		
		
	command_button_init(
	    object_name 				:= CONCAT(prc_path, '_navigate_to_accU_popup_cbtn'),
	    process 					:= prc,
	    CONVERSION_this 			:= navigate_to_accU_popup_cbtn);	
	
	//"toggle" FOR TESTING	
	hmi_graphic_object_status_init(
        object_name         		:= CONCAT(prc_path, '_hmi_toggle_hgos'),
        process             		:= prc,
        CONVERSION_this             := hmi_toggle_hgos);
	
	hmi_graphic_object_status_init(
        object_name         		:= CONCAT(prc_path, '_hmi_brand_status_color_hgos'),
        process             		:= prc,
        CONVERSION_this             := hmi_brand_status_color_hgos);
		
	hmi_graphic_object_status_init(
        object_name         		:= CONCAT(prc_path, '_hmi_brand_status_bad_color_hgos'),
        process             		:= prc,
        CONVERSION_this             := hmi_brand_status_bad_color_hgos);
		
	hmi_graphic_object_status_init(
        object_name         		:= CONCAT(prc_path, '_hmi_accU_step1_on_hgos'),
        process             		:= prc,
        CONVERSION_this             := hmi_accU_step1_on_hgos);
		
	hmi_graphic_object_status_init(
        object_name         		:= CONCAT(prc_path, '_hmi_accU_step1_off_hgos'),
        process             		:= prc,
        CONVERSION_this             := hmi_accU_step1_off_hgos);
		
	hmi_graphic_object_status_init(
        object_name         		:= CONCAT(prc_path, '_hmi_accU_step2_on_hgos'),
        process             		:= prc,
        CONVERSION_this             := hmi_accU_step2_on_hgos);
		
	hmi_graphic_object_status_init(
        object_name         		:= CONCAT(prc_path, '_hmi_accU_step2_off_hgos'),
        process             		:= prc,
        CONVERSION_this             := hmi_accU_step2_off_hgos);
		
	hmi_graphic_object_status_init(
        object_name         		:= CONCAT(prc_path, '_hmi_accU_step3_on_hgos'),
        process             		:= prc,
        CONVERSION_this             := hmi_accU_step3_on_hgos);
		
	hmi_graphic_object_status_init(
        object_name         		:= CONCAT(prc_path, '_hmi_accU_step3_off_hgos'),
        process             		:= prc,
        CONVERSION_this             := hmi_accU_step3_off_hgos);
		
	hmi_graphic_object_status_init(
        object_name         		:= CONCAT(prc_path, '_hmi_accU_step4_on_hgos'),
        process             		:= prc,
        CONVERSION_this             := hmi_accU_step4_on_hgos);
		
	hmi_graphic_object_status_init(
        object_name         		:= CONCAT(prc_path, '_hmi_accU_step4_off_hgos'),
        process             		:= prc,
        CONVERSION_this             := hmi_accU_step4_off_hgos);
		
	hmi_graphic_object_status_init(
        object_name         		:= CONCAT(prc_path, '_hmi_accU_step5_on_hgos'),
        process             		:= prc,
        CONVERSION_this             := hmi_accU_step5_on_hgos);
		
	hmi_graphic_object_status_init(
        object_name         		:= CONCAT(prc_path, '_hmi_accU_step5_off_hgos'),
        process             		:= prc,
        CONVERSION_this             := hmi_accU_step5_off_hgos);
		
	hmi_graphic_object_status_init(
        object_name         		:= CONCAT(prc_path, '_hmi_accU_step6_on_hgos'),
        process             		:= prc,
        CONVERSION_this             := hmi_accU_step6_on_hgos);
		
	hmi_graphic_object_status_init(
        object_name         		:= CONCAT(prc_path, '_hmi_accU_step6_off_hgos'),
        process             		:= prc,
        CONVERSION_this             := hmi_accU_step6_off_hgos);
		
	hmi_graphic_object_status_init(
        object_name         		:= CONCAT(prc_path, '_hmi_accU_step7_on_hgos'),
        process             		:= prc,
        CONVERSION_this             := hmi_accU_step7_on_hgos);
	
	hmi_graphic_object_status_init(
        object_name         		:= CONCAT(prc_path, '_hmi_accU_step7_off_hgos'),
        process             		:= prc,
        CONVERSION_this             := hmi_accU_step7_off_hgos);

	//Change Part EOAT
	hmi_graphic_object_status_init(
        object_name         		:= CONCAT(prc_path, '_hmi_change_part_eoat_red_hgos'),
        process             		:= prc,
        CONVERSION_this             := hmi_change_part_eoat_red_hgos);
		
	hmi_graphic_object_status_init(
        object_name         		:= CONCAT(prc_path, '_hmi_change_part_eoat_green_hgos'),
        process             		:= prc,
        CONVERSION_this             := hmi_change_part_eoat_green_hgos);
		
	hmi_graphic_object_status_init(
        object_name         		:= CONCAT(prc_path, '_hmi_change_part_eoat_blue_hgos'),
        process             		:= prc,
        CONVERSION_this             := hmi_change_part_eoat_blue_hgos);
		
	hmi_graphic_object_status_init(
        object_name         		:= CONCAT(prc_path, '_hmi_change_part_eoat_yellow_hgos'),
        process             		:= prc,
        CONVERSION_this             := hmi_change_part_eoat_yellow_hgos);
	
	hmi_graphic_object_status_init(
        object_name         		:= CONCAT(prc_path, '_hmi_change_part_eoat_white_hgos'),
        process             		:= prc,
        CONVERSION_this             := hmi_change_part_eoat_white_hgos);
		
	hmi_graphic_object_status_init(
        object_name         		:= CONCAT(prc_path, '_hmi_change_part_eoat_black_hgos'),
        process             		:= prc,
        CONVERSION_this             := hmi_change_part_eoat_black_hgos);
		
	hmi_graphic_object_status_init(
        object_name         		:= CONCAT(prc_path, '_hmi_change_part_eoat_orange_hgos'),
        process             		:= prc,
        CONVERSION_this             := hmi_change_part_eoat_orange_hgos);
		
	hmi_graphic_object_status_init(
        object_name         		:= CONCAT(prc_path, '_hmi_change_part_eoat_checkbox_hgos'),
        process             		:= prc,
        CONVERSION_this             := hmi_change_part_eoat_checkbox_hgos);
		
	//Change Part Pusher
	hmi_graphic_object_status_init(
        object_name         		:= CONCAT(prc_path, '_hmi_change_part_pusher_green_hgos'),
        process             		:= prc,
        CONVERSION_this             := hmi_change_part_pusher_green_hgos);
		
	hmi_graphic_object_status_init(
        object_name         		:= CONCAT(prc_path, '_hmi_change_part_pusher_yellow_hgos'),
        process             		:= prc,
        CONVERSION_this             := hmi_change_part_pusher_yellow_hgos);
		
	hmi_graphic_object_status_init(
        object_name         		:= CONCAT(prc_path, '_hmi_change_part_pusher_white_hgos'),
        process             		:= prc,
        CONVERSION_this             := hmi_change_part_pusher_white_hgos);
		
	hmi_graphic_object_status_init(
        object_name         		:= CONCAT(prc_path, '_hmi_change_part_pusher_black_hgos'),
        process             		:= prc,
        CONVERSION_this             := hmi_change_part_pusher_black_hgos);
		
	hmi_graphic_object_status_init(
        object_name         		:= CONCAT(prc_path, '_hmi_change_part_pusher_checkbox_hgos'),
        process             		:= prc,
        CONVERSION_this             := hmi_change_part_pusher_checkbox_hgos);
		
	//Change Part Plate
	hmi_graphic_object_status_init(
        object_name         		:= CONCAT(prc_path, '_hmi_change_part_plate_green_hgos'),
        process             		:= prc,
        CONVERSION_this             := hmi_change_part_plate_green_hgos);
		
	hmi_graphic_object_status_init(
        object_name         		:= CONCAT(prc_path, '_hmi_change_part_plate_yellow_hgos'),
        process             		:= prc,
        CONVERSION_this             := hmi_change_part_plate_yellow_hgos);
		
	hmi_graphic_object_status_init(
        object_name         		:= CONCAT(prc_path, '_hmi_change_part_plate_black_hgos'),
        process             		:= prc,
        CONVERSION_this             := hmi_change_part_plate_black_hgos);
		
	hmi_graphic_object_status_init(
        object_name         		:= CONCAT(prc_path, '_hmi_change_part_plate_checkbox_hgos'),
        process             		:= prc,
        CONVERSION_this             := hmi_change_part_plate_checkbox_hgos);
	
	//Change Part Paddles
	hmi_graphic_object_status_init(
        object_name         		:= CONCAT(prc_path, '_hmi_change_part_paddle_checkbox_hgos'),
        process             		:= prc,
        CONVERSION_this             := hmi_change_part_paddle_checkbox_hgos);
	
		//Change Part In Position
	hmi_graphic_object_status_init(
        object_name         		:= CONCAT(prc_path, '_hmi_in_position_on_hgos'),
        process             		:= prc,
        CONVERSION_this             := hmi_in_position_on_hgos);	
	
	hmi_graphic_object_status_init(
        object_name         		:= CONCAT(prc_path, '_hmi_in_position_off_hgos'),
        process             		:= prc,
        CONVERSION_this             := hmi_in_position_off_hgos);	
	
	process_message_init(
        object_name:= CONCAT(prc_path, '_RFID_read_write_error_msg'),
        behaviour:= MESSAGE_BEHAVIOUR_STATE,
        reset_timeout:= 0,
        disableable:= TRUE,
        individual_reset:= FALSE,
        machine_reaction:= MACHINE_REACTION_NO_STOP, 
        typology:=  MESSAGE_TYPOLOGY_NOT_VISIBLE, 
        process:= prc,
        CONVERSION_this:= RFID_read_write_error_msg);
		
		
	timer_init(
		object_name					:= CONCAT(prc_path, '_brand_change_check_delay_tmr'),
		process						:= prc,
		CONVERSION_this				:= brand_change_check_delay_tmr);
		
			//AAcc U Change in Position indicators
	hmi_graphic_object_status_init(
        object_name         		:= CONCAT(prc_path, '_hmi_in_position_transport_depth_on_hgos'),
        process             		:= prc,
        CONVERSION_this             := hmi_in_position_transport_depth_on_hgos);	
	
	hmi_graphic_object_status_init(
        object_name         		:= CONCAT(prc_path, '_hmi_in_position_transport_depth_off_hgos'),
        process             		:= prc,
        CONVERSION_this             := hmi_in_position_transport_depth_off_hgos);	

	hmi_graphic_object_status_init(
        object_name         		:= CONCAT(prc_path, '_hmi_in_position_shuttle_depth_on_hgos'),
        process             		:= prc,
        CONVERSION_this             := hmi_in_position_shuttle_depth_on_hgos);	
	
	hmi_graphic_object_status_init(
        object_name         		:= CONCAT(prc_path, '_hmi_in_position_shuttle_depth_off_hgos'),
        process             		:= prc,
        CONVERSION_this             := hmi_in_position_shuttle_depth_off_hgos);	
	
		
	hmi_graphic_object_status_init(
        object_name         		:= CONCAT(prc_path, '_hmi_in_position_magazine_ls_depth_on_hgos'),
        process             		:= prc,
        CONVERSION_this             := hmi_in_position_magazine_ls_depth_on_hgos);	
	
	hmi_graphic_object_status_init(
        object_name         		:= CONCAT(prc_path, '_hmi_in_position_magazine_ls_depth_off_hgos'),
        process             		:= prc,
        CONVERSION_this             := hmi_in_position_magazine_ls_depth_off_hgos);	

	hmi_graphic_object_status_init(
        object_name         		:= CONCAT(prc_path, '_hmi_in_position_magazine_os_depth_on_hgos'),
        process             		:= prc,
        CONVERSION_this             := hmi_in_position_magazine_os_depth_on_hgos);	
	
	hmi_graphic_object_status_init(
        object_name         		:= CONCAT(prc_path, '_hmi_in_position_magazine_os_depth_off_hgos'),
        process             		:= prc,
        CONVERSION_this             := hmi_in_position_magazine_os_depth_off_hgos);	

	hmi_graphic_object_status_init(
        object_name         		:= CONCAT(prc_path, '_hmi_in_position_loader_guide_width_on_hgos'),
        process             		:= prc,
        CONVERSION_this             := hmi_in_position_loader_guide_width_on_hgos);	
	
	hmi_graphic_object_status_init(
        object_name         		:= CONCAT(prc_path, '_hmi_in_position_loader_guide_width_off_hgos'),
        process             		:= prc,
        CONVERSION_this             := hmi_in_position_loader_guide_width_off_hgos);	

	hmi_graphic_object_status_init(
        object_name         		:= CONCAT(prc_path, '_hmi_in_position_glue_os_upper_on_hgos'),
        process             		:= prc,
        CONVERSION_this             := hmi_in_position_glue_os_upper_on_hgos);	
	
	hmi_graphic_object_status_init(
        object_name         		:= CONCAT(prc_path, '_hmi_in_position_glue_os_upper_off_hgos'),
        process             		:= prc,
        CONVERSION_this             := hmi_in_position_glue_os_upper_off_hgos);	

	hmi_graphic_object_status_init(
        object_name         		:= CONCAT(prc_path, '_hmi_in_position_glue_os_lower_on_hgos'),
        process             		:= prc,
        CONVERSION_this             := hmi_in_position_glue_os_lower_on_hgos);	
	
	hmi_graphic_object_status_init(
        object_name         		:= CONCAT(prc_path, '_hmi_in_position_glue_os_lower_off_hgos'),
        process             		:= prc,
        CONVERSION_this             := hmi_in_position_glue_os_lower_off_hgos);	

	hmi_graphic_object_status_init(
        object_name         		:= CONCAT(prc_path, '_hmi_in_position_glue_ls_upper_on_hgos'),
        process             		:= prc,
        CONVERSION_this             := hmi_in_position_glue_ls_upper_on_hgos);	
	
	hmi_graphic_object_status_init(
        object_name         		:= CONCAT(prc_path, '_hmi_in_position_glue_ls_upper_off_hgos'),
        process             		:= prc,
        CONVERSION_this             := hmi_in_position_glue_ls_upper_off_hgos);	

	hmi_graphic_object_status_init(
        object_name         		:= CONCAT(prc_path, '_hmi_in_position_glue_ls_lower_on_hgos'),
        process             		:= prc,
        CONVERSION_this             := hmi_in_position_glue_ls_lower_on_hgos);	
	
	hmi_graphic_object_status_init(
        object_name         		:= CONCAT(prc_path, '_hmi_in_position_glue_ls_lower_off_hgos'),
        process             		:= prc,
        CONVERSION_this             := hmi_in_position_glue_ls_lower_off_hgos);	

	hmi_graphic_object_status_init(
        object_name         		:= CONCAT(prc_path, '_hmi_in_position_glue_os_width_on_hgos'),
        process             		:= prc,
        CONVERSION_this             := hmi_in_position_glue_os_width_on_hgos);	
	
	hmi_graphic_object_status_init(
        object_name         		:= CONCAT(prc_path, '_hmi_in_position_glue_os_width_off_hgos'),
        process             		:= prc,
        CONVERSION_this             := hmi_in_position_glue_os_width_off_hgos);	
	
	hmi_graphic_object_status_init(
        object_name         		:= CONCAT(prc_path, '_hmi_in_position_transfer_infeed_depth_on_hgos'),
        process             		:= prc,
        CONVERSION_this             := hmi_in_position_transfer_infeed_depth_on_hgos);	
	
	hmi_graphic_object_status_init(
        object_name         		:= CONCAT(prc_path, '_hmi_in_position_transfer_infeed_depth_off_hgos'),
        process             		:= prc,
        CONVERSION_this             := hmi_in_position_transfer_infeed_depth_off_hgos);	
	
	hmi_graphic_object_status_init(
        object_name         		:= CONCAT(prc_path, '_hmi_in_position_waterfall_on_hgos'),
        process             		:= prc,
        CONVERSION_this             := hmi_in_position_waterfall_on_hgos);	
	
	hmi_graphic_object_status_init(
        object_name         		:= CONCAT(prc_path, '_hmi_in_position_waterfall_off_hgos'),
        process             		:= prc,
        CONVERSION_this             := hmi_in_position_waterfall_off_hgos);	
	
	hmi_graphic_object_status_init(
        object_name         		:= CONCAT(prc_path, '_hmi_in_position_accumulator_depth_on_hgos'),
        process             		:= prc,
        CONVERSION_this             := hmi_in_position_accumulator_depth_on_hgos);	
	
	hmi_graphic_object_status_init(
        object_name         		:= CONCAT(prc_path, '_hmi_in_position_accumulator_depth_off_hgos'),
        process             		:= prc,
        CONVERSION_this             := hmi_in_position_accumulator_depth_off_hgos);	
	
	hmi_graphic_object_status_init(
        object_name         		:= CONCAT(prc_path, '_hmi_in_position_accumulator_conv_depth_on_hgos'),
        process             		:= prc,
        CONVERSION_this             := hmi_in_position_accumulator_conv_depth_on_hgos);	
	
	hmi_graphic_object_status_init(
        object_name         		:= CONCAT(prc_path, '_hmi_in_position_accumulator_conv_depth_off_hgos'),
        process             		:= prc,
        CONVERSION_this             := hmi_in_position_accumulator_conv_depth_off_hgos);	
	hmi_graphic_object_status_init(
        object_name         		:= CONCAT(prc_path, '_hmi_in_position_top_rail_os_width_on_hgos'),
        process             		:= prc,
        CONVERSION_this             := hmi_in_position_top_rail_os_width_on_hgos);	
	
	hmi_graphic_object_status_init(
        object_name         		:= CONCAT(prc_path, '_hmi_in_position_top_rail_os_width_off_hgos'),
        process             		:= prc,
        CONVERSION_this             := hmi_in_position_top_rail_os_width_off_hgos);	
	hmi_graphic_object_status_init(
        object_name         		:= CONCAT(prc_path, '_hmi_in_position_top_rail_ls_width_on_hgos'),
        process             		:= prc,
        CONVERSION_this             := hmi_in_position_top_rail_ls_width_on_hgos);	
	
	hmi_graphic_object_status_init(
        object_name         		:= CONCAT(prc_path, '_hmi_in_position_top_rail_ls_width_off_hgos'),
        process             		:= prc,
        CONVERSION_this             := hmi_in_position_top_rail_ls_width_off_hgos);	
	hmi_graphic_object_status_init(
        object_name         		:= CONCAT(prc_path, '_hmi_in_position_top_rail_depth_on_hgos'),
        process             		:= prc,
        CONVERSION_this             := hmi_in_position_top_rail_depth_on_hgos);	
	
	hmi_graphic_object_status_init(
        object_name         		:= CONCAT(prc_path, '_hmi_in_position_top_rail_depth_off_hgos'),
        process             		:= prc,
        CONVERSION_this             := hmi_in_position_top_rail_depth_off_hgos);	
	hmi_graphic_object_status_init(
        object_name         		:= CONCAT(prc_path, '_hmi_in_position_discharge_os_depth_on_hgos'),
        process             		:= prc,
        CONVERSION_this             := hmi_in_position_discharge_os_depth_on_hgos);	
	
	hmi_graphic_object_status_init(
        object_name         		:= CONCAT(prc_path, '_hmi_in_position_discharge_os_depth_off_hgos'),
        process             		:= prc,
        CONVERSION_this             := hmi_in_position_discharge_os_depth_off_hgos);	
	
	
//HMI graphic object status for machine is ready and enabled for visiblity of read and write button  on the RFID setup screen
	hmi_graphic_object_status_init(
        object_name         		:= CONCAT(prc_path, '_hmi_machine_ready_and_enable_hgos'),
        process             		:= prc,
        CONVERSION_this             := hmi_machine_ready_and_enable_hgos);	

		
	filter_init(
		object_name					:= CONCAT(prc_path, '_horn_on_filter'),
		delay_off_on				:= horn_on_time,
		delay_on_off				:= horn_off_time,
		process						:= prc,
		CONVERSION_this				:= horn_on_filter);
		
	
END_IF

IF objects_running()
THEN
	process_cycle(prc);
	
	command_button_cycle(hmi_toggle_cbtn);
	command_button_cycle(manual_empty_cbtn);
	command_button_cycle(RFID_Setup_read_cbtn);
	command_button_cycle(RFID_Setup_write_cbtn);
	command_button_cycle(brand_change_request_cbtn);
	command_button_cycle(navigate_to_accU_popup_cbtn);
	
	motorization_conditioner_cycle(all_in_position_motcond);
	motorization_conditioner_cycle(eoat_rfid_checked_motcond);
	motorization_conditioner_cycle(loader_pusher_rfid_checked_motcond);
	motorization_conditioner_cycle(loader_plate_rfid_checked_motcond);
	
	digital_check_cycle(stop_machine_for_change_parts_dchk);
	
	filter_cycle(accU_axis_moving_horn_on, horn_on_filter);
END_IF
END_ACTION

ACTION _read_process_image:
command_button_led_set_status(
	status				:= HMI_OBJECT_STATUS_ON, 		
	CONVERSION_this		:= brand_change_request_cbtn);

command_button_led_set_status(
	status				:= HMI_OBJECT_STATUS_ON, 		
	CONVERSION_this		:= navigate_to_accU_popup_cbtn);

brand_change_request_dvr := command_button_is_pressed(brand_change_request_cbtn);
navigate_to_accU_popup_dvr := command_button_is_pressed(navigate_to_accU_popup_cbtn);
END_ACTION

ACTION _read_var_input:
;
END_ACTION

ACTION _set_runtime_properties:
IF navigate_to_accU_popup_dvr
THEN
	navigate_to_accU_popup := FALSE;
	not_in_brand_change := TRUE;
END_IF;
END_ACTION

ACTION _write_output:
;
END_ACTION

ACTION RFID:
IF RFID_reader_list_accuchange <> RFID_reader_list_accuchange_old
THEN
	RFID_Setup_read_value_string := '';
	RFID_Setup_read_value := null_byte;
	RFID_reader_list_accuchange_old := RFID_reader_list_accuchange;
ELSE
	RFID_Setup_read_value_string := BYTE_TO_STRING(RFID_Setup_read_value);
END_IF


IF csp_main_accuChange.RFID_reader_list_accuchange = LOADER_PUSHER_READER
THEN
	loader_plate_in_position := FALSE;
	case_feed_in_position := FALSE;
	closing_os_in_position := FALSE; 
	
	change_part_color := hmi_change_part_pusher_color;
	
	changeover_rfid_read_done := csp_case_loader_pusher.rfid_read_done;
	changeover_rfid_write_done := csp_case_loader_pusher.rfid_write_done;
	changeover_rfid_value := csp_case_loader_pusher.rfid_value;
	changover_rfid_read_write_running := csp_case_loader_pusher.RFID_read_write_running;
	 
	IF csp_case_loader_pusher.rfid_input_bitheader_1.CP
	THEN
		loader_in_position := TRUE;
	END_IF
	 
	
ELSIF csp_main_accuChange.RFID_reader_list_accuchange = CASE_FEED_EOAT_READER
THEN
	loader_in_position := FALSE;
	loader_plate_in_position := FALSE;
	closing_os_in_position := FALSE; 
	
	change_part_color := hmi_change_part_eoat_color;

	changeover_rfid_read_done := csp_case_feed_arm_sensors.rfid_read_done;
	changeover_rfid_write_done := csp_case_feed_arm_sensors.rfid_write_done;
	changeover_rfid_value := csp_case_feed_arm_sensors.rfid_value;
	changover_rfid_read_write_running := csp_case_feed_arm_sensors.RFID_read_write_running;
		
	IF csp_case_feed_arm_sensors.rfid_input_bitheader_1.CP
	THEN
		case_feed_in_position := TRUE;
	END_IF
		 
ELSIF csp_main_accuChange.RFID_reader_list_accuchange = LOADER_GUIDE_PLATE_READER
THEN
	loader_in_position := FALSE;
	case_feed_in_position := FALSE;
	closing_os_in_position := FALSE;
	
	change_part_color := hmi_change_part_plate_color;
	
	changeover_rfid_read_done := csp_case_loader_sensors.rfid_read_done;
	changeover_rfid_write_done := csp_case_loader_sensors.rfid_write_done;
	changeover_rfid_value := csp_case_loader_sensors.rfid_value;
	changover_rfid_read_write_running := csp_case_loader_sensors.RFID_read_write_running;
	
	IF csp_case_loader_sensors.rfid_input_bitheader_1.CP
	THEN
		loader_plate_in_position := TRUE;
	END_IF
		
ELSIF csp_main_accuChange.RFID_reader_list_accuchange = CLOSING_PADDLES_READER
THEN
	loader_in_position := FALSE;
	case_feed_in_position := FALSE;
	loader_plate_in_position := FALSE;
	
	change_part_color := hmi_change_part_paddle_color;

	changeover_rfid_read_done := csp_case_closing.rfid_read_done;
	changeover_rfid_write_done := csp_case_closing.rfid_write_done;
	changeover_rfid_value := csp_case_closing.os_rfid_value;
	changover_rfid_read_write_running := NOT csp_case_closing.rfid_read_done OR NOT csp_case_closing.rfid_write_done;

	IF 	csp_case_closing.os_rfid_input_bitheader_1.CP
		OR csp_case_closing.ls_rfid_input_bitheader_1.CP
	THEN
		closing_os_in_position := TRUE;
	END_IF
	 
END_IF
	
	

//checks all the change parts to see if the selected part is infront of the rfid reader
IF 	loader_in_position
	OR
	case_feed_in_position
	OR
	loader_plate_in_position
	OR
	closing_os_in_position
THEN
	change_part_in_position:= TRUE;
ELSE
	change_part_in_position :=FALSE;	
END_IF

	hmi_graphic_object_set_status(
        status  			:= SEL(change_part_in_position, HMI_OBJECT_STATUS_INVISIBLE, HMI_OBJECT_STATUS_ON),
        CONVERSION_this     := hmi_in_position_on_hgos);
		
	hmi_graphic_object_set_status(
        status  			:= SEL(change_part_in_position, HMI_OBJECT_STATUS_ON, HMI_OBJECT_STATUS_INVISIBLE),
        CONVERSION_this     := hmi_in_position_off_hgos);

		
		
(* READ VALUE FROM RFID TO HIM *)
IF 	command_button_get_actual_value(RFID_Setup_read_cbtn) = HMI_BUTTON_STATUS_ON
	AND machine_is_ready(csp.mch)
THEN
	RFID_read_write_status_next := READ_WRITE_STATUS_START_RFID_READ;
END_IF


IF hmi_toggle_hgos.status = HMI_OBJECT_STATUS_ON
THEN
	enable_write := TRUE;
ELSE
	enable_write := FALSE;
END_IF

(* WRITES VALUE FROM HMI TO RFID *)
IF command_button_get_actual_value(RFID_Setup_write_cbtn) = HMI_BUTTON_STATUS_ON
	AND machine_is_ready(csp.mch)
	AND enable_write
THEN
	RFID_read_write_status_next := READ_WRITE_STATUS_START_RFID_WRITE;
END_IF

(* STATE MACHINE FOR READING AND WRITING TO RFID - ONLY FOR COMMAND BUTTONS*)
CASE RFID_read_write_status OF
	(* READ LOGIC *)
	READ_WRITE_STATUS_START_RFID_READ:
	
		rfid_read_write_running := TRUE;
		RFID_read_write_status_next := READ_WRITE_STATUS_SEND_READ_COMMAND;
		
		
	READ_WRITE_STATUS_SEND_READ_COMMAND:
	
		rfid_reading := TRUE;
		IF changover_rfid_read_write_running
		THEN
			RFID_read_write_status_next := READ_WRITE_STATUS_WAIT_FOR_READ_RESULT;
		END_IF
		
		
	READ_WRITE_STATUS_WAIT_FOR_READ_RESULT:
	
		IF 	rfid_reading
			AND changeover_rfid_read_done (* BE DYNAMIC BASED ON SELECTION - AT TOP *)
		THEN
			RFID_read_write_status_next := READ_WRITE_STATUS_CHECK_READ_RESULT;
		END_IF


	READ_WRITE_STATUS_CHECK_READ_RESULT:
	
		rfid_read_write_running := FALSE;
		rfid_reading := FALSE;
		RFID_Setup_read_value := changeover_rfid_value; (* BE DYNAMIC BASED ON SELECTION - AT TOP *)
		RFID_read_write_status_next := READ_WRITE_STATUS_WAITING;
		
		
	(* WRITE LOGIC *)
	READ_WRITE_STATUS_START_RFID_WRITE:
	
		rfid_read_write_running := TRUE;
		RFID_Setup_write_value := INT_TO_BYTE(RFID_reader_brand_colors);
		RFID_read_write_status_next := READ_WRITE_STATUS_SEND_WRITE_COMMAND;
		
		
	READ_WRITE_STATUS_SEND_WRITE_COMMAND:
	
		rfid_writing := TRUE;
		IF changover_rfid_read_write_running
		THEN
			RFID_read_write_status_next := READ_WRITE_STATUS_WAIT_FOR_WRITE_SUCCESS;
		END_IF
		
		
	READ_WRITE_STATUS_WAIT_FOR_WRITE_SUCCESS:
	
		IF rfid_writing
			AND changeover_rfid_write_done
		THEN
			rfid_read_write_running := FALSE;
			rfid_writing := FALSE;
			
			RFID_read_write_status_next := READ_WRITE_STATUS_WAITING;
		END_IF
		
		
	READ_WRITE_STATUS_WRITE_TO_READ:
	
		RFID_read_write_status_next := READ_WRITE_STATUS_START_RFID_READ;
				
		
	READ_WRITE_STATUS_WAITING:
	
		rfid_read_write_running := FALSE;	
		
		
	READ_WRITE_STATUS_ERROR:
	
		;
	
	
	
END_CASE


(* ADVANCES TO NEXT STEP *)
IF 	NOT RFID_read_write_debug
	OR
	RFID_read_write_one_step	
THEN
	RFID_read_write_status := RFID_read_write_status_next;
	RFID_read_write_one_step := FALSE;
END_IF


(* Connection timeout *)
IF	RFID_read_write_running
	AND NOT RFID_read_write_debug
THEN
	IF	timer_is_expired(RFID_read_write_tmr)
	THEN
		process_message_set(1, RFID_read_write_status, 0, RFID_read_write_error_msg);
	END_IF
ELSE
	timer_restart(10000, RFID_read_write_tmr);
END_IF
END_ACTION

END_PROGRAM

// ---- Application/CSP/Case/Loader/Sensors/csp_case_loader_sensors.TcPOU
(*********************************** G.D S.p.A. - Technical Department ***********************************
============= PROGRAM INFO ============
FOLDER:             TBD
MACHINES INVOLVED:  TBD 

============= DESCRIPTION =============
csp machine declaration

============= REVISIONS ===============
Date		Version	 	Author      	Description             
----------	-------		------------  	--------------------------------------------
2019/04/05 	0000.00	 	M.Grasso		Creation of the PRG

**********************************************************************************************************)
(*$R process_ref := prc; $*)
PROGRAM csp_case_loader_sensors
VAR
	
	prc:												process;
	prc_path:											STRING;
	
	(* RFID *)
	rfid_value:											BYTE;
	rfid_value_to_write:								BYTE;
	
	rfid_input_buffer:									iol_slave_bis00lh_pdo_input;
	rfid_input_bitheader_1:								iol_slave_bis00lh_bitheader_input;
	rfid_input_bitheader_2:								iol_slave_bis00lh_bitheader_input;
			
	rfid_output_buffer:									iol_slave_bis00lh_pdo_output;
	rfid_output_bitheader_1:							iol_slave_bis00lh_bitheader_output;
	rfid_output_bitheader_2:							iol_slave_bis00lh_bitheader_output;
	
	RFID_read_write_status:								csp_case_loader_rfid_status_enum;
	RFID_read_write_status_next:						csp_case_loader_rfid_status_enum;
	RFID_read_write_debug:								BOOL := FALSE;
	RFID_read_write_one_step:							BOOL := FALSE;
	RFID_read_write_running:							BOOL;
	RFID_read_write_tmr:								timer;
	RFID_read_write_error_msg:							message;
	
	rfid_start_toggle:									BOOL := FALSE;
	rfid_shutdown_toggle:								BOOL := FALSE;
	rfid_write_toggle:									BOOL := FALSE;
	rfid_write_done:									BOOL := FALSE;
	rfid_read_toggle:									BOOL := FALSE;
	rfid_read_done:										BOOL := FALSE;
	
END_VAR

_read_var_input();

_object_manager();

IF NOT objects_running()
THEN
	RETURN;	
END_IF

_read_process_image();

_mode_manager();

_set_runtime_properties();

(********************************* BODY *********************************)

IF 	csp_main_accuChange.RFID_reader_list_accuchange = LOADER_GUIDE_PLATE_READER
THEN
	RFID();
END_IF

(************************************************************************)

_handle_messages();

_write_output();

ACTION _handle_messages:
;
END_ACTION

ACTION _handle_process_test:
;
END_ACTION

ACTION _mode_manager:
IF process_mode_req_is_pending(prc)
THEN
    process_apply_mode_req_first_step(prc);
    CASE process_get_mode(prc) OF
        MODE_TO_ABSENT:
			;
        MODE_TO_INACTIVE:
			;
        MODE_TO_TEST:
			;
        MODE_TO_OPERATIONAL:
			;
    END_CASE
    process_apply_mode_req_second_step(prc);
END_IF
END_ACTION

ACTION _object_manager:
IF objects_initialization()
THEN
	sub_process_init(
		object_name					:= 'csp_case_loader_pusher.prc', 
		process						:= csp_case_loader.prc, 
		CONVERSION_this				:= prc);
		
	prc_path 						:= process_get_path(prc);
	
	(* INPUTS *)

	
	
	process_message_init(
        object_name:= CONCAT(prc_path, '_RFID_read_write_error_msg'),
        behaviour:= MESSAGE_BEHAVIOUR_STATE,
        reset_timeout:= 0,
        disableable:= TRUE,
        individual_reset:= FALSE,
        machine_reaction:= MACHINE_REACTION_NO_STOP, //MACHINE_REACTION_STOP_IN_PHASE_ONE,
        typology:=  MESSAGE_TYPOLOGY_NOT_VISIBLE, //MESSAGE_TYPOLOGY_ABNORMAL,
        process:= prc,
        CONVERSION_this:= RFID_read_write_error_msg);
		
END_IF

IF objects_running()
THEN
	process_cycle(prc);
END_IF
END_ACTION

ACTION _read_process_image:
;
END_ACTION

ACTION _read_var_input:
;
END_ACTION

ACTION _set_runtime_properties:
;
END_ACTION

ACTION _write_output:
;
END_ACTION

ACTION RFID:
	(* RMH RFID TEST *)
rfid_input_bitheader_1.CP := rfid_input_buffer.ByteArr[0].0;
rfid_input_bitheader_1.AA := rfid_input_buffer.ByteArr[0].1;
rfid_input_bitheader_1.AE := rfid_input_buffer.ByteArr[0].2;
rfid_input_bitheader_1.AF := rfid_input_buffer.ByteArr[0].3;
rfid_input_bitheader_1.Bit4 := rfid_input_buffer.ByteArr[0].4;
rfid_input_bitheader_1._TO := rfid_input_buffer.ByteArr[0].5;
rfid_input_bitheader_1.HF := rfid_input_buffer.ByteArr[0].6;
rfid_input_bitheader_1.BB := rfid_input_buffer.ByteArr[0].7;

rfid_input_bitheader_2.CP := rfid_input_buffer.ByteArr[0].0;
rfid_input_bitheader_2.AA := rfid_input_buffer.ByteArr[0].1;
rfid_input_bitheader_2.AE := rfid_input_buffer.ByteArr[0].2;
rfid_input_bitheader_2.AF := rfid_input_buffer.ByteArr[0].3;
rfid_input_bitheader_2.Bit4 := rfid_input_buffer.ByteArr[0].4;
rfid_input_bitheader_2._TO := rfid_input_buffer.ByteArr[0].5;
rfid_input_bitheader_2.HF := rfid_input_buffer.ByteArr[0].6;
rfid_input_bitheader_2.BB := rfid_input_buffer.ByteArr[0].7;

rfid_output_buffer.ByteArr[0].0 := rfid_output_bitheader_1.AV ;
rfid_output_buffer.ByteArr[0].1 := rfid_output_bitheader_1.Bit1;
rfid_output_buffer.ByteArr[0].2 := rfid_output_bitheader_1.GR;
rfid_output_buffer.ByteArr[0].3 := rfid_output_bitheader_1.Bit3;
rfid_output_buffer.ByteArr[0].4 := rfid_output_bitheader_1.Bit4;
rfid_output_buffer.ByteArr[0].5 := rfid_output_bitheader_1.KA;
rfid_output_buffer.ByteArr[0].6 := rfid_output_bitheader_1.TI;
rfid_output_buffer.ByteArr[0].7 := rfid_output_bitheader_1.Bit7;

rfid_output_buffer.ByteArr[9].0 := rfid_output_bitheader_2.AV ;
rfid_output_buffer.ByteArr[9].1 := rfid_output_bitheader_2.Bit1;
rfid_output_buffer.ByteArr[9].2 := rfid_output_bitheader_2.GR;
rfid_output_buffer.ByteArr[9].3 := rfid_output_bitheader_2.Bit3;
rfid_output_buffer.ByteArr[9].4 := rfid_output_bitheader_2.Bit4;
rfid_output_buffer.ByteArr[9].5 := rfid_output_bitheader_2.KA;
rfid_output_buffer.ByteArr[9].6 := rfid_output_bitheader_2.TI;
rfid_output_buffer.ByteArr[9].7 := rfid_output_bitheader_2.Bit7;


IF 	rfid_start_toggle
THEN
	rfid_output_bitheader_1.GR := FALSE;
	rfid_output_bitheader_1.KA := FALSE;
	rfid_output_bitheader_1.AV := FALSE;
	rfid_output_bitheader_2.GR := FALSE;
	rfid_output_bitheader_2.KA := FALSE;
	rfid_output_bitheader_2.AV := FALSE;
	
	rfid_start_toggle := FALSE;
END_IF


IF 	rfid_shutdown_toggle
THEN
	rfid_output_bitheader_1.KA := TRUE;
	rfid_output_bitheader_2.KA := TRUE;
	
	IF rfid_input_bitheader_1.HF
		AND rfid_input_bitheader_2.HF
		AND NOT rfid_input_bitheader_1.CP
		AND NOT rfid_input_bitheader_2.CP
	THEN
		rfid_output_bitheader_1.KA := FALSE;
		rfid_output_bitheader_2.KA := FALSE;
		rfid_shutdown_toggle := FALSE;
	END_IF
		
END_IF


IF 	rfid_write_toggle //OR i_rfid_write_from_hmi
THEN	
	rfid_output_buffer.ByteArr[1] := 16#0032;
	rfid_output_buffer.ByteArr[2] := 16#00;
	rfid_output_buffer.ByteArr[3] := 16#00;
	rfid_output_buffer.ByteArr[4] := 16#0001;
	rfid_output_buffer.ByteArr[5] := 16#00;
	rfid_output_buffer.ByteArr[6] := rfid_value_to_write;
	
	rfid_output_bitheader_1.AV := TRUE;
	rfid_output_bitheader_2.AV := TRUE;
	
	IF rfid_input_bitheader_1.AA 
		AND rfid_input_bitheader_2.AA 
		AND rfid_input_bitheader_1.AE
		AND rfid_input_bitheader_2.AE
	THEN
		rfid_output_bitheader_1.AV := FALSE;
		rfid_output_bitheader_2.AV := FALSE;
		rfid_write_toggle := FALSE;
	END_IF
		
END_IF


IF 	rfid_read_toggle 
THEN	
	rfid_output_buffer.ByteArr[1] := 16#0001;
	rfid_output_buffer.ByteArr[2] := 16#00;
	rfid_output_buffer.ByteArr[3] := 16#00;
	rfid_output_buffer.ByteArr[4] := 16#0001;
	rfid_output_buffer.ByteArr[5] := 16#00;
	
	rfid_output_bitheader_1.AV := TRUE;
	rfid_output_bitheader_2.AV := TRUE;
	
	
	IF rfid_input_bitheader_1.AA 
		AND rfid_input_bitheader_2.AA 
		AND rfid_input_bitheader_1.AE
		AND rfid_input_bitheader_2.AE
	THEN
		// SAVE VALUES IN INPUT BUFFER [1...8] - CHECK WITH BRAND FOR WHAT VALUE SHOULD BE PRESENT
		rfid_value := rfid_input_buffer.ByteArr[1];
		rfid_output_bitheader_1.AV := FALSE;
		rfid_output_bitheader_2.AV := FALSE;
		rfid_read_toggle := FALSE;
	END_IF
		
END_IF



(* STATE MACHINE FOR READING AND WRITING TO RFID *)
CASE RFID_read_write_status OF
			
	CSP_CASE_LOADER_RFID_STATUS_START:
	
		IF 	csp_main_accuChange.RFID_read_write_running (* Use this value within brand change to start the check *)
		THEN
			rfid_write_done := FALSE;
			rfid_read_done := FALSE;
			rfid_read_write_running := TRUE;
			RFID_read_write_status_next := CSP_CASE_LOADER_RFID_STATUS_CHECK_READ_WRITE;
		END_IF
		
		
	CSP_CASE_LOADER_RFID_STATUS_CHECK_READ_WRITE:
	
		rfid_start_toggle := TRUE;
		IF 	csp_main_accuChange.RFID_reading (* Use this value also within brand change *)
		THEN
			RFID_read_write_status_next := CSP_CASE_LOADER_RFID_STATUS_READ_START;
		ELSIF csp_main_accuChange.RFID_writing
		THEN
			RFID_read_write_status_next := CSP_CASE_LOADER_RFID_STATUS_WRITE_START;
		END_IF
			
		
		
	(* RFID READ START *)	
	CSP_CASE_LOADER_RFID_STATUS_READ_START:
	
		IF 	rfid_input_bitheader_1.CP
			AND rfid_input_bitheader_2.CP
		THEN
			rfid_read_toggle := TRUE;
			RFID_read_write_status_next := CSP_CASE_LOADER_RFID_STATUS_READ_CHECK_RESULT;
		END_IF
	
	CSP_CASE_LOADER_RFID_STATUS_READ_CHECK_RESULT:
	
		IF 	NOT rfid_read_toggle 
		THEN
			RFID_read_write_status_next := CSP_CASE_LOADER_RFID_STATUS_READ_DONE;
		END_IF
		
	CSP_CASE_LOADER_RFID_STATUS_READ_DONE:
	
		rfid_read_done := TRUE;
		rfid_read_write_running := FALSE;
		RFID_read_write_status_next := CSP_CASE_LOADER_RFID_STATUS_WAITING;
		
		
	(* RFID WRITING START *)
	CSP_CASE_LOADER_RFID_STATUS_WRITE_START:
	
		rfid_value_to_write := csp_main_accuChange.RFID_Setup_write_value;
		
		IF 	rfid_input_bitheader_1.CP
			AND rfid_input_bitheader_2.CP
		THEN
			rfid_write_toggle := TRUE;
			RFID_read_write_status_next := CSP_CASE_LOADER_RFID_STATUS_WAIT_WRITE;
		END_IF
		
	CSP_CASE_LOADER_RFID_STATUS_WAIT_WRITE:
	
		IF 	NOT rfid_write_toggle
		THEN	
			RFID_read_write_status_next := CSP_CASE_LOADER_RFID_STATUS_WRITE_DONE;
		END_IF
		
	CSP_CASE_LOADER_RFID_STATUS_WRITE_DONE:
	
		rfid_write_done := TRUE;
		rfid_read_write_running := FALSE;
		RFID_read_write_status_next := CSP_CASE_LOADER_RFID_STATUS_WAITING;
		
	
	CSP_CASE_LOADER_RFID_STATUS_WAITING:
	
		IF 	csp_main_accuchange.RFID_read_write_running
		THEN
			RFID_read_write_status_next := CSP_CASE_LOADER_RFID_STATUS_START;
		END_IF
		
END_CASE


(* ADVANCES TO NEXT STEP *)
IF 	NOT RFID_read_write_debug
	OR
	RFID_read_write_one_step	
THEN
	RFID_read_write_status := RFID_read_write_status_next;
	RFID_read_write_one_step := FALSE;
END_IF


(* Connection timeout *)
IF	RFID_read_write_running
	AND NOT RFID_read_write_debug
THEN
	IF	timer_is_expired(RFID_read_write_tmr)
	THEN
		rfid_start_toggle := TRUE;
		process_message_set(1, RFID_read_write_status, 0, RFID_read_write_error_msg);
	END_IF
ELSE
	timer_restart(10000, RFID_read_write_tmr);
END_IF
END_ACTION

END_PROGRAM

// ---- Application/CSP/Case/Loader/csp_case_loader.TcPOU
(*********************************** G.D S.p.A. - Technical Department ***********************************
============= PROGRAM INFO ============
FOLDER:             TBD
MACHINES INVOLVED:  TBD 

============= DESCRIPTION =============
csp machine declaration

============= REVISIONS ===============
Date		Version	 	Author      	Description             
----------	-------		------------  	--------------------------------------------
2019/04/05 	0000.00	 	M.Grasso		Creation of the PRG

**********************************************************************************************************)
(*$R process_ref := prc; $*)
PROGRAM csp_case_loader
VAR
	
	prc:											process;
	prc_path:										STRING;
	load_request:                                   BOOL:=FALSE;
 	case_at_loading_sr:								INT:=26;
	product_at_loading_sr:							INT:=25;
	
	shift_test1: 									BOOL;
	test_1: 										BOOL := FALSE;
	
	follower_clear_test: 							BOOL := FALSE;
	follower_tolerance: 							INT := 16;
	follower_clear: 								BOOL := FALSE;
	horizontal_clear: 								BOOL := FALSE;
	load_ready_at_loader: 							BOOL := FALSE;
	cases_primed:									BOOL := FALSE;
	case_at_loader:									BOOL := FALSE;
	
	dry_cycle_on:									BOOL := FALSE;
	dry_cycle_turned_off_clear_prime:				BOOL;
	
	case_removed_at_feed:							BOOL := FALSE;
	case_removed_at_feed_cbtn:						command_button;

	case_removed_at_loader_cbtn:                    command_button;
    case_removed_at_loader:                         BOOL := FALSE;
	
	phasing_order_done:								BOOL;
	phase_leading_minor:							BOOL;
	phase_loader_guides:							BOOL;
	phase_loader_pusher:							BOOL;
	phase_follower:									BOOL;
	
	phasing_status:									csp_case_phasing_enum;
	phasing_status_next:							csp_case_phasing_enum;
		
	phase_conditions:								BOOL;
	
	
	cases_primed_ph:								phase;
	cases_primed_check_deg:							LREAL := 353;
	
	
	Clear_out_cartons_at_Loader: 					message;
	bypass_new_phase: 								BOOL := TRUE;
	
	phase_timer:									TON;
	phase_timer_enable:								BOOL := FALSE;
	phase_timer_limit:								TIME := T#20S;
END_VAR

_read_var_input();

_object_manager();

IF NOT objects_running()
THEN
	RETURN;	
END_IF

_read_process_image();

_mode_manager();

_set_runtime_properties();

(********************************* BODY *********************************)
IF 	shift_register_step_has_status_item(
		step_id := 25,
		status_bits_to_be_true := ITEM_CASE_FEED,
		status_bits_to_be_false := 0,
		CONVERSION_this :=csp_case_main_statistics.sr) 
THEN
	cases_primed := TRUE;
ELSE 
	cases_primed := FALSE;
END_IF

IF 	shift_register_step_has_status_item(
		step_id := 26,
		status_bits_to_be_true := ITEM_CASE_FEED,
		status_bits_to_be_false := 0,
		CONVERSION_this :=csp_case_main_statistics.sr) 
THEN
	case_at_loader := TRUE;
ELSE 
	case_at_loader := FALSE;
END_IF

(* AT RESET IT TURNS ON THE FOLLOWER IS CLEAR TO START*)
IF 	machine_get_reset_edge(CSP.mch)
THEN
	follower_clear_test := TRUE;
END_IF


(* VERIFIES LOADER IS CLEAR AND WILL NOT RUN *)
IF 	follower_clear_test
	OR ABS(csp_transfer_crosspusher_follower.axis.actual_position - csp_transfer_crosspusher_follower.slave_scaling) < follower_tolerance
THEN
	follower_clear := TRUE;
ELSE
	follower_clear := FALSE;
END_IF	

IF 	csp_transfer_crosspusher_horizontal.axis.actual_position > -1  
THEN
	horizontal_clear := TRUE;
ELSE
	horizontal_clear := FALSE;
END_IF


//IF phase_edge(csp_case_loader_virtualMaster.load_check_ph)
IF 	csp_transfer_upstacker.stack_at_loader (* STACK HAS BEEN PUSHED FROM UPSTACKER TO LOAD *)
//AND horizontal_clear(* FOLLOWER AT LOAD *)
//AND follower_Clear
	AND NOT csp_transfer_crosspusher_sensors.reject_stack (* NOT REJECT STACK *)
	AND NOT csp_transfer_crosspusher_sensors.stack_fail (* NOT STACK FAIL *)
	AND NOT csp_transfer_crosspusher_sensors.no_load_bool.status (* NOT NO LOAD *)
THEN
	load_ready_at_loader := TRUE; // STACK AT LOADER AND HORIZONTAL AND FOLLOWER CLEAR
ELSE
	load_ready_at_loader := FALSE;
END_IF


(* PRIMES CASES - KEEPS PRIMED IF IN JOG *)
IF 	jog_manager_is_jog_axis_active(JOG_LIST_CSP_CASE_VIRTUAL, csp_main_jogManager.jog_manager_virtual)	
THEN
	shift_register_set_status_item(
		step_id                 :=  25,
		status_bits_to_set      :=  ITEM_CASE_FEED,
		status_bits_to_reset    :=  0,
		CONVERSION_this         :=  csp_case_main_statistics.sr);//cases_primed := TRUE;
END_IF


(* MANUAL REMOVAL OF CASES PRIMED*)
IF 	command_button_is_pressed(case_removed_at_feed_cbtn) 
THEN
	case_removed_at_feed := TRUE;
ELSE
	case_removed_at_feed := FALSE;
END_IF


(* CONDITIONS TO CLEAR CASES PRIMED *)
IF 	case_removed_at_feed
//OR csp_case_transport_virtualMaster.STOP_FOR_REJECT
//OR csp_case_transport_virtualMaster.Bad_case_detected
//OR dry_cycle_turned_off_clear_prime //MOVED TO CSP_CASE_MAIN_STATISTICS TO CLEAR OUT WHOLE SR!
//OR csp_case_feed_arm_sensors.mispick_count >= 1 //AMR 3_16_2021
	OR process_message_is_on(csp_case_virtualMaster.runout_complete)
	OR message_is_on(csp_case_feed_arm_sensors.Mispicked_Case_aem)	
	OR csp_main_accuChange.Brand_Change_Occurred
THEN
	shift_register_set_default_step(25,csp_case_main_statistics.sr);//cases_primed := FALSE;
	dry_cycle_turned_off_clear_prime := FALSE;
END_IF




(* TOGGLES ON DRY CYCLE TO SET FOR BIT CLEARING *)
IF 	csp_case_main_services.dry_cycle_mode
THEN
	dry_cycle_on := TRUE;
END_IF

IF 	dry_cycle_on
	AND NOT csp_case_main_services.dry_cycle_mode
THEN
	dry_cycle_turned_off_clear_prime := TRUE;
	dry_cycle_on := FALSE;
END_IF



(* PHASE EDGE FOR CASE VIRTUAL TO DETERMINE CASES PRIMED *)
phase_set_data(
	phase				:= cases_primed_check_deg,
	delay				:= 0,			
	max_compensation	:= 0,			
	CONVERSION_this		:= cases_primed_ph);



IF 	shift_register_step_has_status_item(
		step_id := product_at_loading_sr,
		status_bits_to_be_true := ITEM_HAS_TRANSFER_LOAD_BUILD_COMPLETE, // ITEM_PRESENT,
		status_bits_to_be_false := 0,
		CONVERSION_this :=csp_case_main_statistics.sr)
THEN
	shift_test1 := TRUE;
ELSE
	shift_test1 := FALSE;
END_IF


IF  shift_register_step_has_status_item(
   		step_id := case_at_loading_sr,
    	status_bits_to_be_true :=  ITEM_HAS_LS_LOWER_FLAP + ITEM_HAS_LS_UPPER_FLAP + ITEM_HAS_OS_LOWER_FLAP + ITEM_HAS_OS_UPPER_FLAP,
    	status_bits_to_be_false := 0,
    	CONVERSION_this :=csp_case_main_statistics.sr)
		
	AND load_ready_at_loader
	AND NOT csp_case_loader_virtualMaster.product_loaded 
	AND NOT test_1
THEN
    load_request :=TRUE;
ELSE
    load_request :=FALSE;
END_IF

IF 	(csp_case_transport_virtualMaster.axis.actual_modulo_position = 358//csp_case_loader_virtualMaster.At_Reject_product_loaded 
	AND csp_case_transport_virtualMaster.stop_for_reject)
THEN
	test_1 := TRUE;
ELSIF csp_case_feed.Feed_request
THEN
	test_1 := FALSE;
END_IF
	
(* Axes engaged for jog management *) 
jog_manager_set_all_slave_axis_engaged(
	index					:= JOG_LIST_CSP_CASE_loader_VIRTUAL, 
	all_slave_axis_engaged	:= csp_case_loader_virtualMaster.loader_slaves_cammed,						 	
	CONVERSION_this			:= csp_main_jogManager.jog_manager_virtual);

	
	
(* LOGIC TO HANDLE PHASING SEQUENCE OF TRAILING MINOR CLOSER LS, LOADER GUIDES UP/DOWN, LOADER PUSHER, CROSSPUSHER FOLLOWER *)

(* TURNS OFF PHASING ORDER DONE IF ANY AXES BECOME NOT CAM ENGAGED *)
(*IF NOT axis_is_cam_engaged(csp_case_fc_ls_upper_leadingMinorCloser.axis)
AND NOT axis_is_cam_engaged(csp_case_loader_guide_downstream.axis)
AND NOT axis_is_cam_engaged(csp_case_loader_guide_upstream.axis)
AND NOT axis_is_cam_engaged(csp_case_loader_pusher.axis)
AND NOT axis_is_cam_engaged(csp_transfer_crosspusher_follower.axis)
AND NOT bypass_new_phase*)
IF 	csp.o_machine_is_stopped
	AND NOT bypass_new_phase
THEN
	phasing_order_done := FALSE;
	
	phase_leading_minor := FALSE;
	phase_loader_guides := FALSE;
	phase_loader_pusher := FALSE;
	phase_follower := FALSE;
	//phasing_status := CSP_CASE_PHASING_START;
		
END_IF

IF 	NOT csp_main_accuChange.machine_size_complete //bypass logic during size change
THEN
	bypass_new_phase := TRUE;
ELSE
	;//bypass_new_phase := FALSE;
END_IF

IF 	bypass_new_phase
THEN
	phasing_order_done := TRUE;
	phasing_status := CSP_CASE_PHASING_DONE;
END_IF



phase_conditions := 
	process_is_ready(prc)
	AND
	process_subtree_is_ready(prc)
	AND
	NOT phasing_order_done;
	
(*Initialize phase timer*)	
phase_timer(IN:= phase_timer_enable, PT:= phase_timer_limit);

(*If time is elapsed, end phasing as to not get stuck and hang up other parts*)
IF 	phase_timer.Q
THEN
	phasing_status := CSP_CASE_PHASING_DONE;
END_IF
	
(* Exit condition *)
IF 	NOT phase_conditions
	OR csp_case_main_services_pushbuttons.reset_pressed
	OR csp_transfer_main_services_pushbuttons.reset_pressed
THEN
	phasing_status_next := CSP_CASE_PHASING_ERROR;
	phasing_status := phasing_status_next;	
END_IF


phasing_status := phasing_status_next;


(* MANUAL REMOVAL OF CASES AT LOADER*)
IF 	command_button_is_pressed(case_removed_at_loader_cbtn)
THEN
	shift_register_set_default_step(26,csp_case_main_statistics.sr);//case_at_loader := FALSE;
	IF 	csp_transfer_upstacker.stack_in_case_at_loader
	THEN
		case_removed_at_loader := TRUE;
	END_IF
END_IF


IF 	case_removed_at_loader
	AND NOT case_at_loader
	AND csp_transfer_upstacker.stack_at_loader
	AND csp_case_loader_pusher.axis.actual_position > 700
THEN
    process_message_set(1,1,1, Clear_out_cartons_at_Loader);
    case_removed_at_loader := FALSE;
end_if

 

IF 	NOT csp_case_main_safety_guards.sis.is_safely_closed //or NOT csp_transfer_main_safety_guards.sis.is_safely_closed
    AND
    process_message_is_on(Clear_out_cartons_at_Loader)
THEN
	process_message_reset(Clear_out_cartons_at_Loader);
END_IF
	
(************************************************************************)

_handle_messages();

_write_output();

ACTION _handle_messages:
;
END_ACTION

ACTION _handle_process_test:
;
END_ACTION

ACTION _mode_manager:
IF process_mode_req_is_pending(prc)
THEN
    process_apply_mode_req_first_step(prc);
    CASE process_get_mode(prc) OF
        MODE_TO_ABSENT:
			;
        MODE_TO_INACTIVE:
			;
        MODE_TO_TEST:
			;
        MODE_TO_OPERATIONAL:
			;
    END_CASE
    process_apply_mode_req_second_step(prc);
END_IF
END_ACTION

ACTION _object_manager:
IF objects_initialization()
THEN
    sub_process_init(
        object_name                    := 'csp_case_loader.prc', 
        process                        := csp_case.prc, 
        CONVERSION_this                := prc);
        
    prc_path                         := process_get_path(prc);
    

    command_button_init(
        object_name                 := CONCAT(prc_path, '_case_removed_at_feed_cbtn'),
        process                     := prc,
        CONVERSION_this             := case_removed_at_feed_cbtn);    
    
    command_button_init(
        object_name                 := CONCAT(prc_path, '_case_removed_at_loader_cbtn'),
        process                     := prc,
        CONVERSION_this             := case_removed_at_loader_cbtn);    
        
    phase_init(
        object_name                 := CONCAT(prc_path, '_cases_primed_ph'),
        phase                         := 0,    //Set at runtime!
        delay                         := 0,
        max_compensation             := 0,
        generator                     := csp_case_feed_virtualMaster.case_fed_phgen, // CHANGE TO LOADER VIRTUAL PHGEN
        process                     := prc,
        CONVERSION_this             := cases_primed_ph);
    
    process_message_init(
        object_name                    := CONCAT(prc_path, '_Clear_out_cartons_at_Loader'), 
        behaviour                    := MESSAGE_BEHAVIOUR_STATE,
        reset_timeout                := 0,
        disableable                    := TRUE,
        individual_reset            := FALSE,
        machine_reaction            := MACHINE_REACTION_EMERGENCY_STOP,
        typology                    := MESSAGE_TYPOLOGY_ABNORMAL,
        process                        := prc,
        CONVERSION_this                := Clear_out_cartons_at_Loader);
    
    
END_IF

IF objects_running()
THEN
    process_cycle(prc);
    
    phase_cycle(cases_primed_ph);
    
    command_button_cycle(case_removed_at_feed_cbtn);
    command_button_cycle(case_removed_at_loader_cbtn);
END_IF
END_ACTION

ACTION _read_process_image:
;
END_ACTION

ACTION _read_var_input:
;
END_ACTION

ACTION _set_runtime_properties:
;
END_ACTION

ACTION _write_output:
;
END_ACTION

END_PROGRAM

// ---- Application/CSP/Case/Main/statistics/csp_case_main_statistics.TcPOU
(*********************************** G.D S.p.A. - Technical Department ***********************************
============= PROGRAM INFO ============
FOLDER:             TBD
MACHINES INVOLVED:  TBD 

============= DESCRIPTION =============
WU exit shift register

============= REVISIONS ===============
Date		Version	 	Author      	Description             
----------	-------		------------  	--------------------------------------------
2019/04/24 	0000.00	 	G.Cera 			Creation of the PRG

**********************************************************************************************************)
(*$R
	process_ref := prc;
$*)
PROGRAM csp_case_main_statistics
VAR
	prc:											process;
	prc_path:										STRING;
	
	sr:												shift_register;
	sr_id:											shift_register_id;
	
	logsect:										log_section;
	
	(* Machine emptying *)	
	number_of_products:								INT;
	counter:										DINT;
	shift_first_step_to_check:						DINT;
	shift_last_step_to_check:						DINT;	
	is_empty:										BOOL;
	reject_shift_array:								ARRAY [0..30] OF BOOL; 
	number_of_rejects: 								INT;
	counter1:										DINT;
	amr_step_shift: 								INT;
	AMR_TEST_1: 									BOOL;
	ResetSRDefault: 								BOOL;
	i:												DINT;
	number_of_boxes: 								INT;
	counter2:										DINT;
	boxes_shift_array:								ARRAY [0..30] OF BOOL; 
	SHIFT_case_at_feed: 							BOOL;
	SHIFT_case_at_loader: 							BOOL;
	SHIFT_case_at_closing: 							BOOL;
	SHIFT_case_at_discharge: 						BOOL;
	SHIFT_case_at_unused: 							BOOL;

	Set_case_at_feed: 								BOOL;
	Set_case_at_loader: 							BOOL;
END_VAR

VAR CONSTANT
	SHIFT_LAST_STEP:								INT := 29;
END_VAR

_read_var_input();

_object_manager();

IF NOT objects_running()
THEN
	RETURN;	
END_IF

_read_process_image();

_mode_manager();

CASE process_get_mode(prc) of
	MODE_ABSENT,
	MODE_INACTIVE:
		is_empty := TRUE;	
	
		RETURN;
	MODE_TEST:
		_handle_process_test();
END_CASE

_set_runtime_properties();

(********************************* BODY *********************************)
(* Manage of the machine emptying *)
shift_first_step_to_check :=
	shift_register_get_first_step(sr);
	
shift_last_step_to_check :=
	SHIFT_LAST_STEP;

number_of_products:= 0;
FOR counter:= shift_first_step_to_check TO shift_last_step_to_check BY 1 DO
	IF	shift_register_step_has_status_item(
			step_id:= counter,
			status_bits_to_be_true:= ITEM_CASE_FEED,
			status_bits_to_be_false:= 0,
			CONVERSION_this:= sr)
	THEN
		number_of_products:= number_of_products + 1;
	END_IF
END_FOR

IF	number_of_products <> 0
THEN
	is_empty:= FALSE;
ELSE
	is_empty:= TRUE;
END_IF

IF csp_case_main_services.dry_cycle_mode
THEN
	log_section_disable(logsect);
ELSE
	log_section_enable(logsect);
END_IF

number_of_rejects:= 0;
FOR counter1:= shift_first_step_to_check TO shift_last_step_to_check BY 1 DO
	IF	shift_register_step_has_any_reject_reason(
			step_id:= counter1,
			CONVERSION_this:= sr)
	THEN
		number_of_rejects:= number_of_rejects + 1;
		reject_shift_array[counter1] := 1; (* A 1 indicates a shift step with reject status *)
	ELSE
		reject_shift_array[counter1] := 0;(* A 0 indicates a shift step with no reject *)
	END_IF
END_FOR

(*Clears shift register when the cleanout mode has been completed *)
IF process_message_is_on(csp_case_virtualMaster.runout_complete)
	OR csp_transfer_upstacker.dry_cycle_ftrig.Q
	OR csp_main_accuChange.Brand_Change_Occurred
	OR ResetSRDefault
THEN
	FOR i := shift_first_step_to_check TO shift_last_step_to_check BY 1 DO
	shift_register_set_default_step(i,sr);
	END_FOR
END_IF

(*Resets shift to default state of blank (empty) *)
IF AMR_TEST_1
THEN
	shift_register_set_default_step(amr_step_shift,sr);
END_IF

number_of_boxes:= 0;
FOR counter2:= shift_first_step_to_check TO shift_last_step_to_check BY 1 DO
	IF	shift_register_step_has_status_item(
			step_id:= counter2,
			status_bits_to_be_true:= ITEM_CASE_FEED,
			status_bits_to_be_false:= 0,
			CONVERSION_this:= sr)
	THEN
		number_of_boxes:= number_of_boxes + 1;
		boxes_shift_array[counter2] := 1; (* A 1 indicates a shift step case status *)
	ELSE
		boxes_shift_array[counter2] := 0;(* A 0 indicates a shift step with *)
	END_IF
END_FOR

IF	shift_register_step_has_status_item(
			step_id:= 25,
			status_bits_to_be_true:= ITEM_CASE_FEED,
			status_bits_to_be_false:= 0,
			CONVERSION_this:= sr)
THEN
	SHIFT_case_at_feed := TRUE;
ELSE
	SHIFT_case_at_feed := FALSE;	
END_IF

IF	shift_register_step_has_status_item(
			step_id:= 26,
			status_bits_to_be_true:= ITEM_CASE_FEED,
			status_bits_to_be_false:= 0,
			CONVERSION_this:= sr)
THEN
	SHIFT_case_at_loader := TRUE;
ELSE
	SHIFT_case_at_loader := FALSE;	
END_IF

IF	shift_register_step_has_status_item(
			step_id:= 27,
			status_bits_to_be_true:= ITEM_CASE_FEED,
			status_bits_to_be_false:= 0,
			CONVERSION_this:= sr)
THEN
	SHIFT_case_at_closing := TRUE;
ELSE
	SHIFT_case_at_closing := FALSE;	
END_IF

IF	shift_register_step_has_status_item(
			step_id:= 28,
			status_bits_to_be_true:= ITEM_CASE_FEED,
			status_bits_to_be_false:= 0,
			CONVERSION_this:= sr)
THEN
	SHIFT_case_at_discharge := TRUE;
ELSE
	SHIFT_case_at_discharge := FALSE;	
END_IF

IF	shift_register_step_has_status_item(
			step_id:= 29,
			status_bits_to_be_true:= ITEM_CASE_FEED,
			status_bits_to_be_false:= 0,
			CONVERSION_this:= sr)
THEN
	SHIFT_case_at_unused := TRUE;
ELSE
	SHIFT_case_at_unused := FALSE;	
END_IF

(* Sets case at feed true for step 25 *)
IF 	Set_case_at_feed
THEN
	shift_register_set_status_item(
		step_id                 :=  25,
		status_bits_to_set      :=  ITEM_CASE_FEED,
		status_bits_to_reset    :=  0,
		CONVERSION_this         :=  csp_case_main_statistics.sr);
	Set_case_at_feed := FALSE;
END_IF

(* Sets case at feed true for step 26 *)
IF 	Set_case_at_loader
THEN
	shift_register_set_status_item(
		step_id                 :=  26,
		status_bits_to_set      :=  ITEM_CASE_FEED,
		status_bits_to_reset    :=  0,
		CONVERSION_this         :=  csp_case_main_statistics.sr);
	Set_case_at_loader := FALSE;
END_IF
(************************************************************************)

_handle_messages();

_write_output();

ACTION _handle_messages:
;
END_ACTION

ACTION _handle_process_test:
;
END_ACTION

ACTION _mode_manager:
IF process_mode_req_is_pending(prc)
THEN
    process_apply_mode_req_first_step(prc);
    CASE process_get_mode(prc) OF
        MODE_TO_ABSENT:
			;
        MODE_TO_INACTIVE:
			;
        MODE_TO_TEST:
			;
        MODE_TO_OPERATIONAL:
			;
    END_CASE
    process_apply_mode_req_second_step(prc);
END_IF
END_ACTION

ACTION _object_manager:
IF objects_initialization()
THEN
	sub_process_init(
		object_name						:= 'csp_case_main_statistics.prc', 
		process							:= csp_case_feed.prc, 
		CONVERSION_this					:= prc);
		
	prc_path 							:= process_get_path(prc);
	
	shift_register_init(
		object_name						:=	CONCAT(prc_path, '_sr'), 
		enable							:=	TRUE,
		shift_phase						:=	1,
		first_step						:=	2,
		startup_item_state_info			:=	ITEM_ABSENT,
		equipment						:=	SHIFT_REGISTER_NO_EQUIPMENT,
		number_of_equipments			:=	1,
		generator						:=	csp_case_transport_virtualMaster.transport_vm_phgen,
		process							:=	prc,
		CONVERSION_this					:=	sr);
		
	log_section_init(
		object_name						:= CONCAT(prc_path, '_logsect'),
		last_step						:= 29,
		log_enable						:= TRUE, 
		shift_register					:= sr, 
		process							:= prc, 
		CONVERSION_this					:= logsect);

END_IF

IF objects_running()
THEN
	process_cycle(prc);
END_IF
END_ACTION

ACTION _read_process_image:
;
END_ACTION

ACTION _read_var_input:
;
END_ACTION

ACTION _set_runtime_properties:
;
END_ACTION

ACTION _write_output:
;
END_ACTION

END_PROGRAM

// ---- Application/CSP/Transfer/Upstacker/csp_transfer_upstacker.TcPOU
(*********************************** G.D S.p.A. - Technical Department ***********************************
============= PROGRAM INFO ============
FOLDER:             TBD
MACHINES INVOLVED:  TBD 

============= DESCRIPTION =============
csp machine declaration

============= REVISIONS ===============
Date		Version	 	Author      	Description             
----------	-------		------------  	--------------------------------------------
2019/04/05 	0000.00	 	M.Grasso		Creation of the PRG

**********************************************************************************************************)
(*$R process_ref := prc; $*)
PROGRAM csp_transfer_upstacker
VAR
	
	prc:											process;
	prc_path:										STRING;
	
	move_request:									BOOL;
	
	debug_active_bool:								BOOL := FALSE;
	debug_active_clear:								BOOL := FALSE;
	dry_cycle_ftrig:                                F_TRIG;
	cleanout_mode_ftrig:                            F_TRIG;
	
	stack_count:									INT := 0; (*$M $*)
	stack_made:										BOOL := FALSE; (*$M $*)
	stack_on_way_to_loader:							BOOL := FALSE; (*$M $*)
	stack_at_loader:								BOOL := FALSE; (*$M $*)
	clear_pos_stack_at_loader:						LREAL := 800;
	
	stack_in_case_at_loader:						BOOL := FALSE; (*$M $*)
	stack_in_case_at_loader_boolean:				boolean;
	
	stack_count_remainder:							INT;
	
	stack_made_test:								BOOL := FALSE;
	
	test_loader_enable:								BOOL := TRUE;
	test_loader_timer:								timer;
	test_loader_stroke_time:						UINT := 150;
	
	cam_check_ph:									phase;
	phgen:											phase_generator;
	
	
	stack_removed_from_upstack:						BOOL := FALSE;
	stack_removed_from_upstack_cbtn:				command_button;
	
	
	First_cycle_after_dry: 							BOOL;
END_VAR

_read_var_input();

_object_manager();

IF NOT objects_running()
THEN
	RETURN;	
END_IF

_read_process_image();

_mode_manager();

_set_runtime_properties();

(********************************* BODY *********************************)

phase_set_data(
	phase				:= csp_transfer_upstacker_sensors.BACKSTOP_CHECK_DEG, //CAM_CHECK_DEG
	delay				:= 0,			
	max_compensation	:= 0,			
	CONVERSION_this		:= cam_check_ph);
	

(* COUNTS STACK BASED OFF OF CURRENT UPSTACKER CAM AND TRANSFER VIRTUAL CROSSING ZERO *)
IF 	phase_edge(csp_transfer_upstacker_sensors.count_stack_ph)
	AND ((digital_input_is_active(csp_transfer_upstacker_sensors.carton_backstop_di) OR csp_transfer_upstacker_sensors.debug_active) OR (csp_transfer_upstacker_sensors.cleanout_one_stack_timeout AND csp_main_motorization.empty_command))  //AMR
	AND (csp_transfer_upstacker_virtualMaster.active_cam = FORWARD_CAM
	OR csp_transfer_upstacker_virtualMaster.active_cam = TRANSFER_UPSTACKER_VIRTUAL_START_CAM)
THEN
	stack_count := stack_count + 1;
END_IF


(* IF AN UPSTACKER MOTOR FAULTS AFTER THE COUNT STACK PHASE EDGE, A STACK COUNT WILL BE REMOVED *)
IF 	csp_transfer_accumulator_virtualMaster.axis.actual_position > csp_transfer_upstacker_sensors.COUNT_STACK_PHASE_CHECK
	AND 
	(
		NOT axis_is_ok(TRUE, csp_transfer_upstacker_upstream.axis)
		OR
		NOT axis_is_ok(TRUE, csp_transfer_upstacker_downstream.axis)
	)
	AND stack_count > 0
THEN
	stack_count := stack_count - 1;
END_IF


